// TwinCAT 3 PLC project V3_5
// Company: AQUAERO
// libraries:
//   Recipe Management,newest,System
//   VisuSymbols,3.5.10.0,System
//   Tc2_BA, * (Beckhoff Automation GmbH)
//   Tc2_Math, * (Beckhoff Automation GmbH)
//   Tc2_ModbusSrv, * (Beckhoff Automation GmbH)
//   Tc2_Standard, * (Beckhoff Automation GmbH)
//   Tc2_Standard, * (Beckhoff Automation GmbH)
//   Tc2_System, * (Beckhoff Automation GmbH)
//   Tc2_System, * (Beckhoff Automation GmbH)
//   Tc2_TcpIp, * (Beckhoff Automation GmbH)
//   Tc2_Utilities, * (Beckhoff Automation GmbH)
//   Tc3_BA_Common, * (Beckhoff Automation GmbH)
//   Tc3_Module, * (Beckhoff Automation GmbH)
//   Tc3_Module, * (Beckhoff Automation GmbH)
//   VisuDialogs, * (System)
// project tree:
//   Data types/ E_ClientServerSteps.TcDUT, ST_FrameFifoEntry.TcDUT
//   Global Variables/ GVL.TcGVL, GVL_1.TcGVL, TwinCAT_Configuration.TcGVL, Variablen_Konfiguration.TcGVL
//   / GlobalImagePool.TcGIPO (not stored), GlobalTextList.TcGTLO, Recipe Manager.TcRMO (not stored), Standard.TcTTO, Visualization Manager.TcVMO (not stored), VISU_TASK.TcTTO
//   POUs/ Average.TcPOU, Controller.TcPOU, FB_Blink.TcPOU, FB_PeerToPeer.TcPOU, SCL_MAIN.TcPOU, Meine_HYST.TcPOU
//   POUs/Helper POUs/ FB_FrameFifo.TcPOU, FB_LogFifo.TcPOU
//   Visualizations/ ImagePool.TcIPO (not stored), PID.TcVIS (not stored), Main.TcVIS (not stored), PID_alt.TcVIS (not stored), Layout.TcVIS (not stored), Heatreg.TcVIS (not stored), Sensors.TcVIS (not stored), Service.TcVIS (not stored), Testseite1.TcVIS (not stored), FRAME.TcVIS (not stored)
// real-time tasks:
//   TASK Standard: cycle T#10ms, priority 20, ADS port 350
//   TASK VISU_TASK: cycle T#200000us, priority 30, ADS port 351
//   TASK VISU_TASK1: cycle T#1ms, priority 1, ADS port 352

CONFIGURATION V3_5
    RESOURCE PLC ON TwinCAT3
        TASK Standard(INTERVAL := T#10ms, PRIORITY := 20);
        TASK VISU_TASK(INTERVAL := T#200000us, PRIORITY := 30);
        PROGRAM SCL_MAIN WITH Standard : SCL_MAIN;
        PROGRAM VisuElems_Visu_Prg WITH VISU_TASK : VisuElems.Visu_Prg;
    END_RESOURCE
END_CONFIGURATION

// ---- Data types/E_ClientServerSteps.TcDUT
TYPE E_ClientServerSteps :
(
	eUDP_STATE_IDLE		:= 0,
	eUDP_STATE_CREATE_START,
	eUDP_STATE_CREATE_WAIT,
	eUDP_STATE_SEND_START,
	eUDP_STATE_SEND_WAIT,
	eUDP_STATE_RECEIVE_START,
	eUDP_STATE_RECEIVE_WAIT,
	eUDP_STATE_CLOSE_START,
	eUDP_STATE_CLOSE_WAIT,
	eUDP_STATE_ERROR
);
END_TYPE

// ---- Data types/ST_FrameFifoEntry.TcDUT
TYPE ST_FrameFifoEntry :
STRUCT
	stRemoteAddr 	: ST_SockAddr;(* Remote address. String containing an (Ipv4) Internet Protocol dotted address and port number. *)
	sMessage		: T_MaxString;	(* UDP packet data *)
	r_Write_Example : REAL:=999;
	
	
	
END_STRUCT
END_TYPE

// ---- Global Variables/GVL.TcGVL






{attribute 'Tc2GvlVarNames'}
VAR_GLOBAL


(*_____________________________________________________________________________________________________________________________*)


	(*Ab hier Sind Globale Variablen Aquaero*)



	Main_Relais  AT%Q*:BOOL;
	Reset_M_R: BOOL;
	Set_M_R: BOOL;
	Reset_D_M: BOOL;
	Set_D_M: BOOL;
	Switch_OFF_Mainswitch: BOOL;









	(*Not-Aus Relais*)
	Feedback_Mainswitch AT%I*:BOOL;	(*EIngang NotAus-Relais*)
	Start_Mainswitch: BOOL;
	OUT_Mainswitch AT%Q*:BOOL;	(*Pulsausgang NotAus-Relais*)
	Mainswitch_OK: BOOL;
	ERROR_Mainswitch: BOOL;
	RESET_ERROR_Mainswitch: BOOL;
	Cabinet_OK: BOOL;
	VDC_24_OK AT%I*:BOOL;	(*Netzgerät OK*)

	VDC_OK: BOOL;











(* MODBUS *)

	mb_Input_Coils        : ARRAY [0..255] OF BOOL;
	mb_Output_Coils       : ARRAY [0..255] OF BOOL;
	mb_Input_Registers    : ARRAY [0..255] OF WORD;
	mb_Output_Registers   : ARRAY [0..255] OF WORD;



	Register_IN1: INT;
	Register_IN2: INT;
	Register_IN3: INT;
	Register_IN4: INT;
	Register_IN5: INT;
	Register_IN6: INT;
	Register_IN7: INT;
	Register_IN8: INT;
	Register_IN9: INT;
	Register_IN10: INT;



(*Regler_Kompressor Scroll*)


	Activate_controller_comp: BOOL;
	fRegelgroesse_comp: REAL;
	fSollwert_comp: REAL;				(*Ist zurzeit auf Sollert Dampfkammerdruck bezogen, der Kompressor ist das Stellglied*)
	fManual_controller_comp: REAL;
	Set_Manual_controller_comp: BOOL;
	fStellwert_comp: REAL;
	Reset_Controller_comp:BOOL;
	fKP_Controller_comp: REAL;
	fKI_Controller_comp: REAL;




(*Regler_Kompressor Klauenkolbenkomp.*)

	Activate_controller_Primaer_comp: BOOL;
	fRegelgroesse_Primaer_comp: REAL;
	fSollwert_Primaer_comp: REAL;
	fManual_controller_Primaer_comp: REAL;
	Set_Manual_controller_Primaer_comp: BOOL;
	fStellwert_Primaer_comp: REAL;
	Reset_Controller_Primaer_comp:BOOL;
	fKP_Controller_Primaer_comp: REAL:=1;
	fKI_Controller_Primaer_comp: REAL:=0.1;



(*Regler_Umdampfventi*)


	Activate_controller_V_Umdampf: BOOL;
	fRegelgroesse_V_Umdampf: REAL;
	fSollwert_V_Umdampf: REAL;				(*Ist zurzeit auf Sollert Dampfkammerdruck bezogen, der Kompressor ist das Stellglied*)
	fManual_controller_V_Umdampf: REAL;
	Set_Manual_controller_V_Umdampf: BOOL;
	fStellwert_V_Umdampf: REAL;
	Reset_Controller_V_Umdampf:BOOL;
	fKP_Controller_V_Umdampf: REAL;
	fKI_Controller_V_Umdampf: REAL;



(*Regler_Ventilator*)

	Activate_controller_Venti:  BOOL;
	fRegelgroesse_Venti: REAL;
	fSollwert_Venti: REAL;				(*Ist zurzeit auf Sollert Dampfkammerdruck bezogen, der Kompressor ist das Stellglied*)
	fManual_controller_Venti: REAL;
	Set_Manual_controller_Venti: BOOL;
	fStellwert_Venti: REAL;
	Reset_Controller_Venti:BOOL;
	fKP_Controller_Venti: REAL;
	fKI_Controller_Venti: REAL;




(*Regler_Nadelventil Swagelock*)



	Activate_controller_Needlevalve: BOOL;
	fRegelgroesse_NV: REAL;
	fSollwert_NV: REAL;				(*Ist zurzeit auf Sollert Dampfkammerdruck bezogen, der Kompressor ist das Stellglied*)
	fManual_controller_NV: REAL;
	Set_Manual_controller_NV: BOOL;
	fStellwert_NV: REAL;
	Reset_Controller_NV:BOOL;
	fKP_Controller_NV: REAL;
	fKI_Controller_NV: REAL;

	Sollwert_OUT_NV :INT;
	Istwert_IN_NV :INT;





	C_ADS: INT;
	C_DES: INT;




(*Ab hier: Sensorik und Aktorik des neuen Monstartors, oberhalb sind teils nicht verwendete Variablen!!*)





	T_Vor_WT_IN AT%I* : INT;
	T_Vor_WT:REAL;
	T_Vor_WT_Visu:REAL;
	T_nach_WT_IN AT%I* : INT;
	T_nach_WT:REAL;
	T_nach_WT_Visu:REAL;

	T_HE_Einduesung_Oben_IN AT%I* : INT;
	T_HE_Einduesung_Oben:REAL;
	T_HE_Einduesung_Oben_Visu:REAL;

	T_HE_Einduesung_Unten_IN AT%I* : INT;
	T_HE_Einduesung_Unten:REAL;
	T_HE_Einduesung_Unten_Visu:REAL;

	T_Einduesung_Unten_IN AT%I* : INT;
	T_Einduesung_Unten:REAL;
	T_Einduesung_Unten_Visu:REAL;

	T_Einduesung_Oben_IN AT%I* : INT;
	T_Einduesung_Oben:REAL;
	T_Einduesung_Oben_Visu:REAL;


	T_Absaugung_Oben_IN AT%I* : INT;
	T_Absaugung_Oben:REAL;
	T_Absaugung_Oben_Visu:REAL;

	T_Absaugung_Unten_IN AT%I* : INT;
	T_Absaugung_Unten:REAL;
	T_Absaugung_Unten_Visu:REAL;


	T_Vor_UmdampfLuefter_IN AT%I* : INT;
	T_Vor_UmdampfLuefter:REAL;
	T_Vor_UmdampfLuefter_Visu:REAL;

	T_Komp_Auslass_IN AT%I* : INT;
	T_Komp_Auslass:REAL;
	T_Komp_Auslass_Visu:REAL;

	T_Komp_Einlass_IN AT%I* : INT;
	T_Komp_Einlass:REAL;
	T_Komp_Einlass_Visu:REAL;


	T_Kond_Auslass_IN AT%I* : INT;
	T_Kond_Auslass:REAL;
	T_Kond_Auslass_Visu:REAL;

	T_DK_Oben_IN AT%I* : INT;
	T_DK_Oben:REAL;
	T_DK_Oben_Visu:REAL;

	T_DK_Mitte_IN AT%I* : INT;
	T_DK_Mitte:REAL;
	T_DK_Mitte_Visu:REAL;

	T_DK_Unten_IN AT%I* : INT;
	T_DK_Unten:REAL;
	T_DK_Unten_Visu:REAL;
	
	
	
	
	

	T_Mat_Auslass1_IN AT%I* : INT;
	T_Mat_Auslass1:REAL;
	T_Mat_Auslass1_Visu:REAL;
	T_Mat_Auslass2_IN AT%I* : INT;
	T_Mat_Auslass2:REAL;
	T_Mat_Auslass2_Visu:REAL;
	T_Mat_Auslass3_IN AT%I* : INT;
	T_Mat_Auslass3:REAL;
	T_Mat_Auslass3_Visu:REAL;
	T_Mat_Auslass4_IN AT%I* : INT;
	T_Mat_Auslass4:REAL;
	T_Mat_Auslass4_Visu:REAL;
	

	T_Mat_Auslass5_IN AT%I* : INT;
	T_Mat_Auslass5:REAL;
	T_Mat_Auslass5_Visu:REAL;
	T_Mat_Auslass6_IN AT%I* : INT;
	T_Mat_Auslass6:REAL;
	T_Mat_Auslass6_Visu:REAL;
	T_Mat_Auslass7_IN AT%I* : INT;
	T_Mat_Auslass7:REAL;
	T_Mat_Auslass7_Visu:REAL;
	T_Mat_Auslass8_IN AT%I* : INT;
	T_Mat_Auslass8:REAL;
	T_Mat_Auslass8_Visu:REAL;
	
	
	
	
	
	
	
	
	
	
	
	

	T_Komp_Gehaeuse_IN AT%I* : INT;
	T_Komp_Gehaeuse:REAL;
	T_Komp_Gehaeuse_Visu:REAL;


	T_DK_Band_oben1_IN AT%I* : INT;
	T_DK_Band_oben1:REAL;
	T_DK_Band_oben1_Visu:REAL;
	T_DK_Band_oben2_IN  : INT;
	T_DK_Band_oben2:REAL;
	T_DK_Band_oben2_Visu:REAL;
	T_DK_Band_oben3_IN AT%I* : INT;
	T_DK_Band_oben3:REAL;
	T_DK_Band_oben3_Visu:REAL;


	T_DK_Band_unten1_IN AT%I* : INT;
	T_DK_Band_unten1:REAL;
	T_DK_Band_unten1_Visu:REAL;
	T_DK_Band_unten2_IN : INT;
	T_DK_Band_unten2:REAL;
	T_DK_Band_unten2_Visu:REAL;
	T_DK_Band_unten3_IN AT%I* : INT;
	T_DK_Band_unten3:REAL;
	T_DK_Band_unten3_Visu:REAL;
	

	T_DK_Steigband1_IN AT%I* : INT;
	T_DK_Steigband1:REAL;
	T_DK_Steigband1_Visu:REAL;
	T_DK_Steigband2_IN AT%I* : INT;
	T_DK_Steigband2:REAL;
	T_DK_Steigband2_Visu:REAL;
	T_DK_Steigband3_IN AT%I* : INT;
	T_DK_Steigband3:REAL;
	T_DK_Steigband3_Visu:REAL;
	T_DK_Steigband4_IN AT%I* : INT;
	T_DK_Steigband4:REAL;
	T_DK_Steigband4_Visu:REAL;

	
	
	
	
	
	


	Temp_Heatmatt1_IN  AT%I* : INT;
	Temp_Heatmatt2_IN  AT%I* : INT;
	Temp_Heatmatt3_IN  AT%I* : INT;
	Temp_Heatmatt4_IN  AT%I* : INT;
	Temp_Heatmatt5_IN  AT%I* : INT;
	Temp_Heatmatt6_IN  AT%I* : INT;
	Temp_Heatmatt7_IN  AT%I* : INT;
	Temp_Heatmatt8_IN  AT%I* : INT;
	Temp_Heatmatt9_IN  AT%I* : INT;
	Temp_Heatmatt10_IN  AT%I* : INT;


	

	Temp_Heatmatt1 : INT;
	Temp_Heatmatt2 : INT;
	Temp_Heatmatt3 : INT;
	Temp_Heatmatt4 : INT;
	Temp_Heatmatt5 : INT;
	Temp_Heatmatt6 : INT;
	Temp_Heatmatt7 : INT;
	Temp_Heatmatt8 : INT;
	Temp_Heatmatt9 : INT;
	Temp_Heatmatt10 : INT;

	Temp_compressor_Self : INT;




	P_Vor_WT_IN AT%I* : INT;
	P_Vor_WT:REAL;
	P_Vor_WT_Visu:REAL;


	P_Durchfluss_IN  : INT;
	P_Durchfluss:REAL;
	P_Durchfluss_Visu:REAL;



	P_Komp_Einlass_IN AT%I* : INT;
	P_Komp_Einlass:REAL;
	P_Komp_Einlass_Visu:REAL;


	P_Komp_Auslass_IN AT%I* : INT;
	P_Komp_Auslass:REAL;
	P_Komp_Auslass_Visu:REAL;


	W_Kond_Wasser_IN AT%I* : INT;
	W_Kond_Wasser:REAL;
	W_Kond_Wasser_Visu:REAL;



	O2_IN AT%I* : INT;
	O2:REAL;
	O2_Visu:REAL;

	

	PTC_IN:BOOL;
	Motor_HOT:BOOL;

	Switch_Heat_group1:BOOL;
	Switch_Heat_group2:BOOL;
	Switch_Heat_group3:BOOL;
	Start_Auto_Export: BOOL;
	Start_Auto_Export_OUT: BOOL;




	(* Diverses (teils noch von älterenb Programmfunktionen*)

	Pulse2_set_manu:BOOL;
	Enable_Pulsgen2 :BOOL;
	T_Pulstime_Pulsegen2: INT:=3;
	T_HI_Pulsegen2: INT:=20;
	Valve_YB7:BOOL;












(*Strom und Energiemessung*)


	(*Current_IN_HZE_Auffangbecken_L1 AT%I*:INT;
	Current_IN_HZE_Auffangbecken_L2 AT%I*:INT;
	Current_IN_HZE_Auffangbecken_L3 AT%I*:INT;*)

	Current_IN_HEAT_Reg_1 AT%I*:INT;
	Current_IN_HEAT_Reg_2 AT%I*:INT;
	Current_IN_HEAT_Reg_3 AT%I*:INT;
	Current_IN_HEAT_Reg_4 AT%I*:INT;
	Current_IN_HEAT_Reg_5 AT%I*:INT;
	Current_IN_HEAT_Reg_6 AT%I*:INT;
	Current_IN_HEAT_Reg_7 AT%I*:INT;
	Current_IN_HEAT_Reg_8 AT%I*:INT;
	Current_IN_Compressor_L1 AT%I*:INT;
	Current_IN_Compressor_L2 AT%I*:INT;
	Current_IN_Compressor_L3 AT%I*:INT;
	Current_IN_SteamFan_L1 AT%I*:INT;
	Current_IN_SteamFan_L2 AT%I*:INT;
	Current_IN_SteamFan_L3 AT%I*:INT;
	Current_IN_Fan_L1 AT%I*:INT;
	Current_IN_Fan_L2 AT%I*:INT;
	Current_IN_Fan_L3 AT%I*:INT;
	Current_IN_Complete_L1 AT%I*:INT;
	Current_IN_Complete_L2 AT%I*:INT;
	Current_IN_Complete_L3 AT%I*:INT;



	

	Current_OUT_SteamVenti_L1:REAL;
	Current_OUT_SteamVenti_L2:REAL;
	Current_OUT_SteamVenti_L3:REAL;
	Current_OUT_HEAT_Reg_1:REAL;
	Current_OUT_HEAT_Reg_2:REAL;
	Current_OUT_HEAT_Reg_3:REAL;
	Current_OUT_HEAT_Reg_4:REAL;
	Current_OUT_HEAT_Reg_5:REAL;
	Current_OUT_HEAT_Reg_6:REAL;
	Current_OUT_HEAT_Reg_7:REAL;
	Current_OUT_HEAT_Reg_8:REAL;






	Current_OUT_Compressor_L1 :REAL;
	Current_OUT_Compressor_L2 :REAL;
	Current_OUT_Compressor_L3 :REAL;

	Current_OUT_AdsorbtionsVenti_L1 :REAL;
	Current_OUT_AdsorbtionsVenti_L2 :REAL;
	Current_OUT_AdsorbtionsVenti_L3 :REAL;
	Current_OUT_Fan_L1:REAL;
	Current_OUT_Fan_L2 :REAL;
	Current_OUT_Fan_L3:REAL;
	Current_OUT_Complete_L1 :REAL;
	Current_OUT_Complete_L2 :REAL;
	Current_OUT_Complete_L3 :REAL;






	(*Energy_IN_HZE_Auffangbecken_L1 AT%I*:INT;
	Energy_IN_HZE_Auffangbecken_L2 AT%I*:INT;
	Energy_IN_HZE_Auffangbecken_L3 AT%I*:INT;*)

	(*
	Energy_IN_HEAT_Reg_1 AT%I*:INT;
	Energy_IN_HEAT_Reg_2 AT%I*:INT;
	Energy_IN_HEAT_Reg_3 AT%I*:INT;
	Energy_IN_HEAT_Reg_4 AT%I*:INT;
	Energy_IN_Compressor_L1 AT%I*:INT;
	Energy_IN_Compressor_L2 AT%I*:INT;
	Energy_IN_Compressor_L3 AT%I*:INT;
	Energy_IN_SteamFan_L1 AT%I*:INT;
	Energy_IN_SteamFan_L2 AT%I*:INT;
	Energy_IN_SteamFan_L3 AT%I*:INT;
	Energy_IN_Fan_L1 AT%I*:INT;
	Energy_IN_Fan_L2 AT%I*:INT;
	Energy_IN_Fan_L3 AT%I*:INT;
	Energy_IN_Complete_L1 AT%I*:INT;
	Energy_IN_Complete_L2 AT%I*:INT;
	Energy_IN_Complete_L3 AT%I*:INT;*)

	
	
	

	Energy_OUT_HZE_Auffangbecken_L1:REAL;
	Energy_OUT_HZE_Auffangbecken_L2:REAL;
	Energy_OUT_HZE_Auffangbecken_L3:REAL;

	Energy_OUT_HEAT_Reg_1:REAL;
	Energy_OUT_HEAT_Reg_2:REAL;
	Energy_OUT_HEAT_Reg_3:REAL;
	Energy_OUT_HEAT_Reg_4:REAL;
	Energy_OUT_HEAT_Reg_5:REAL;
	Energy_OUT_HEAT_Reg_6:REAL;
	Energy_OUT_HEAT_Reg_7:REAL;
	Energy_OUT_HEAT_Reg_8:REAL;





	Energy_OUT_Compressor_L1 :REAL;
	Energy_OUT_Compressor_L2 :REAL;
	Energy_OUT_Compressor_L3 :REAL;
	Energy_OUT_SteamFan_L1 :REAL;
	Energy_OUT_SteamFan_L2 :REAL;
	Energy_OUT_SteamFan_L3 :REAL;
	Energy_OUT_Fan_L1:REAL;
	Energy_OUT_Fan_L2 :REAL;
	Energy_OUT_Fan_L3:REAL;
	Energy_OUT_Complete_L1 :REAL;
	Energy_OUT_Complete_L2 :REAL;
	Energy_OUT_Complete_L3 :REAL;






(*_________Frequence_Converter_Groups and controls*)

	Compressor_ON AT%Q* : BOOL;
	Compressor_Switch_ON AT%Q* : BOOL;
	Compressor_OK AT%I* : BOOL;
	Compressor_Circuit_breaker AT%I* : BOOL;
	Compressor_Setpoint_OUT AT%Q* : INT;
	Setpoint_Compressor_IN: INT;
	Setpoint_Compressor_Auto: INT;
	Setpoint_Compressor_Visu: INT;
	Compressor_Actual_Turn_IN AT%I* : INT;
	Compressor_Actual_Turn: REAL;
	Limit_Temp_Compressor: INT:=100;
	Temp_compressor_OK: BOOL;
	T_Ueberwachung_scroll_comp AT%I* : INT;


	Compressor_cooling  : BOOL;
	Compressor_cooling_manu  : BOOL;
	Compressor_cooling_auto : BOOL;
	Compressor_Switch_ON_Manu: BOOL;
	Compressor_ON_Manu: BOOL;
	Compressor_PT100_value AT%I* : INT;
	Compressor_PT100_error AT%I* : BOOL;






	(*
	PRIMAER_Comp_ON AT%Q* : BOOL;
	PRIMAER_Comp_OK AT%I* : BOOL;
	PRIMAER_Comp_Setpoint_OUT AT%Q* : INT;
	Setpoint_PRIMAER_Comp_IN: INT;
	Setpoint_PRIMAER_Comp_Auto: INT;
	Setpoint_PRIMAER_Comp_Visu: INT;
	PRIMAER_Comp_Actual_Turn_IN AT%I* : INT;
	PRIMAER_Comp_Actual_Turn: REAL;
	Temp_PRIMAER_Comp_OK: BOOL;
	PRIMAER_Comp_Switch_ON_Manu: BOOL;
	PRIMAER_Comp_ON_Manu: BOOL;
	*)



	Fan_ON  : BOOL;
	Fan_OK  : BOOL;
	Setpoint_Fan_Auto: INT;
	Setpoint_Fan_Visu: INT;
	Setpoint_Fan_OUT  : INT;
	Setpoint_Fan_IN: INT;
	Fan_Actual_Turn_IN  : INT;
	Fan_Actual_Turn  : REAL;
	FAN_Switch_ON  : BOOL;
	FAN_Switch_ON_Manu: BOOL;
	FAN_ON_Manu: BOOL;



	SteamFan_ON AT%Q* : BOOL;
	SteamFan_OK :BOOL ;(* Zurzeit nicht einlesbar AT%I* : BOOL;*)
	Setpoint_SteamFan_Auto: INT;
	Setpoint_SteamFan_Visu: INT;
	Setpoint_SteamFan_OUT AT%Q* : INT;
	Setpoint_SteamFan_IN: INT;
	SteamFan_Actual_Turn_IN AT%I* : INT;
	SteamFan_Actual_Turn  : REAL;
	SteamFAN_Switch_ON AT%Q* : BOOL;
	SteamFAN_Switch_ON_manu:BOOL;
	SteamFan_ON_manu:BOOL;
	Setpoint_SteamFan_manu:INT;
	SteamFan_PTC_IN AT%I* : BOOL;
	SteamFan_PTC_Error AT%I* : BOOL;



	M_Belts_ON AT%Q* : BOOL;
	M_Belts_OK AT%I* : BOOL;
	Setpoint_M_Belts_Auto: INT;
	Setpoint_M_Belts_Visu: INT;
	Setpoint_M_Belts_OUT AT%Q* : INT;
	Setpoint_M_Belts_IN: INT;
	M_Belts_Actual_Turn_IN AT%I* : INT;
	M_Belts_Actual_Turn  : REAL;
	M_Belts_Switch_ON AT%Q* : BOOL;
	M_Belts_Switch_ON_Manu: BOOL;
	M_Belts_ON_Manu: BOOL;
	Activate_controller_M_Belts:BOOL;
	fStellwert_M_Belts:REAL;


	M_Belt_Feeder_ON AT%Q* : BOOL;
	M_Belt_Feeder_OK AT%I* : BOOL;
	Setpoint_M_Belt_Feeder_Auto: INT;
	Setpoint_M_Belt_Feeder_Visu: INT;
	Setpoint_M_Belt_Feeder_OUT AT%Q* : INT;
	Setpoint_M_Belt_Feeder_IN: INT;
	M_Belt_Feeder_Actual_Turn_IN AT%I* : INT;
	M_Belt_Feeder_Actual_Turn  : REAL;
	M_Belt_Feeder_Switch_ON AT%Q* : BOOL;
	M_Belt_Feeder_Switch_ON_Manu: BOOL;
	M_Belt_Feeder_ON_Manu: BOOL;
	Activate_controller_M_Belt_Feeder:BOOL;
	fStellwert_M_Belt_Feeder:REAL;


	Steamgenerator : BOOL;
	Steamgenerator_manu: BOOL;
	Steamgenerator_auto: BOOL;



(*_________Frequence_Converter_Groups AND controls*)
















	(*OUT_______BOOL____________*)



	

	V_Dampf_nach_Komp  AT%Q* : BOOL ;
	V_Dampf_nach_Komp_negiert  AT%Q* : BOOL;
	V_Nach_WT  AT%Q* : BOOL;
	V_Entlueftung_1 AT%Q* : BOOL;
	V_Entlueftung_2 AT%Q* : BOOL;
	V_Global_Res_3 AT%Q* : BOOL;
	V_Global_Res_4 AT%Q* : BOOL;
	V_Global_Res_5 AT%Q* : BOOL;




	Heizelement_Auffangbecken_Mainswitch: BOOL;



	Heat_matt_Group1_1_4 :BOOL;
	Heat_matt_Group2_5_8 :BOOL;
	Heat_matt_Group3_9_10: BOOL;

	Heat_matt1 : BOOL;
	Heat_matt2 : BOOL;
	Heat_matt3 : BOOL;
	Heat_matt4 : BOOL;
	Heat_matt5 : BOOL;
	Heat_matt6 : BOOL;
	Heat_matt7 : BOOL;
	Heat_matt8 : BOOL;
	Heat_matt9 : BOOL;
	Heat_matt10 : BOOL;


	Heat_Matt1_OK_for_heat:BOOL;
	Heat_Matt2_OK_for_heat:BOOL;
	Heat_Matt3_OK_for_heat:BOOL;
	Heat_Matt4_OK_for_heat:BOOL;
	Heat_Matt5_OK_for_heat:BOOL;
	Heat_Matt6_OK_for_heat:BOOL;
	Heat_Matt7_OK_for_heat:BOOL;
	Heat_Matt8_OK_for_heat:BOOL;
	Heat_Matt9_OK_for_heat:BOOL;
	Heat_Matt10_OK_for_heat:BOOL;
	Heat_Matt11_OK_for_heat: BOOL;




	HEAT_Reg_Mainswitch_OUT : BOOL;


	HEAT_Reg_1_OUT AT%Q* : BOOL;
	HEAT_Reg_2_OUT AT%Q* : BOOL;
	HEAT_Reg_3_OUT AT%Q* : BOOL;
	HEAT_Reg_4_OUT AT%Q* : BOOL;
	HEAT_Reg_5_OUT AT%Q* : BOOL;
	HEAT_Reg_6_OUT AT%Q* : BOOL;
	HEAT_Reg_7_OUT AT%Q* : BOOL;
	HEAT_Reg_8_OUT AT%Q* : BOOL;






	V_Nach_WT_negiert: BOOL;
	V_Wasserauslass_negiert: BOOL;
	V_Entlueftung_1_negiert: BOOL;
	V_Global_Res_5_negiert: BOOL;
	V_Global_Res_4_negiert: BOOL;
	V_Global_Res_3_negiert: BOOL;
	V_Entlueftung_2_negiert: BOOL;







	(*AUTO_____________BOOL_____________*)




	(*neuere Aktoren von MS2*)

	V_Dampf_nach_Komp_auto : BOOL:=FALSE;
	V_Nach_WT_auto:BOOL:=FALSE;
	V_Entlueftung_1_auto : BOOL;
	V_Entlueftung_2_auto : BOOL:=FALSE;
	V_Global_Res_3_auto : BOOL:=FALSE;
	V_Global_Res_4_auto : BOOL:=FALSE;
	V_Global_Res_5_auto : BOOL;



	Heat_matt1_auto: BOOL;
	Heat_matt2_auto: BOOL;
	Heat_matt3_auto: BOOL;
	Heat_matt4_auto: BOOL;
	Heat_matt5_auto: BOOL;
	Heat_matt6_auto: BOOL;
	Heat_matt8_auto: BOOL;
	Heat_matt7_auto:BOOL;
	Heat_matt9_auto: BOOL;
	Heat_matt10_auto: BOOL;

	Heat_matt_Group1_1_4_auto: BOOL;
	Heat_matt_Group2_5_8_auto: BOOL;
	Heat_matt_Group3_9_10_auto: BOOL;


	HEAT_Reg_Mainswitch_Auto:BOOL;

	HEAT_Reg_1_Auto: BOOL;
	HEAT_Reg_2_Auto: BOOL;
	HEAT_Reg_3_Auto: BOOL;
	HEAT_Reg_4_Auto: BOOL;
	HEAT_Reg_5_Auto: BOOL;
	HEAT_Reg_6_Auto: BOOL;
	HEAT_Reg_7_Auto: BOOL;
	HEAT_Reg_8_Auto: BOOL;







	(*MANU____________BOOL___________*)


	(*neuere Aktoren von MS2*)


	V_Dampf_nach_Komp_manu : BOOL:=FALSE;
	V_Nach_WT_manu : BOOL:=FALSE;
	V_Entlueftung_1_manu : BOOL:=FALSE;
	V_Entlueftung_2_manu : BOOL;
	V_Global_Res_3_manu : BOOL;
	V_Global_Res_4_manu: BOOL:=FALSE;
	V_Global_Res_5_manu : BOOL;




	Heat_matt1_manu: BOOL;
	Heat_matt2_manu: BOOL;
	Heat_matt3_manu: BOOL;
	Heat_matt4_manu: BOOL;
	Heat_matt5_manu: BOOL;
	Heat_matt6_manu: BOOL;
	Heat_matt7_manu: BOOL;
	Heat_matt8_manu: BOOL;
	Heat_matt9_manu: BOOL;
	Heat_matt10_manu: BOOL;



	HEAT_Reg_Mainswitch_Manu:BOOL;


	HEAT_Reg_1_Manu: BOOL;
	HEAT_Reg_2_Manu: BOOL;
	HEAT_Reg_3_Manu: BOOL;
	HEAT_Reg_4_Manu: BOOL;
	HEAT_Reg_5_Manu: BOOL;
	HEAT_Reg_6_Manu: BOOL;
	HEAT_Reg_7_Manu: BOOL;
	HEAT_Reg_8_Manu: BOOL;





(*________________________________________________________________ENDE_MANU_Vars________________________________*)


















	V_Entlueftung_1_Reset:BOOL;
	V_Entlueftung_2_Reset:BOOL;
	V_Global_Res_3_Reset:BOOL;
	V_Global_Res_4_Reset:BOOL;
	V_Global_Res_5_Reset:BOOL;
	V_Dampf_nach_Komp_Reset:BOOL;
	V_Nach_WT_Reset:BOOL;


	V_Entlueftung_1_String:STRING;
	V_Entlueftung_2_String:STRING;
	V_Global_Res_3_String:STRING;
	V_Global_Res_4_String:STRING;
	V_Global_Res_5_String:STRING;
	V_Dampf_nach_Komp_String:STRING;
	V_NACH_WT_String:STRING;


	V_Entlueftung_1_Reset_Sequence:BOOL;
	V_Entlueftung_2_Reset_Sequence:BOOL;
	V_Global_Res_3_Reset_Sequence:BOOL;
	V_Global_Res_4_Reset_Sequence:BOOL;
	V_Global_Res_5_Reset_Sequence:BOOL;
	V_Dampf_nach_Komp_Reset_Sequence:BOOL;
	V_NACH_WT_Reset_Sequence:BOOL;


	V_Entlueftung_1_Sequence:BOOL;
	V_Entlueftung_2_Sequence:BOOL;
	V_Global_Res_3_Sequence:BOOL;
	V_Global_Res_4_Sequence:BOOL;
	V_Global_Res_5_Sequence:BOOL;
	V_Dampf_nach_Komp_Sequence:BOOL;
	V_NACH_WT_Sequence:BOOL;



	VE_K2_71:BOOL;
	VE_K2_73:BOOL;











	LED_RED_OUT AT%Q* :BOOL;
	LED_RED_VISU: BOOL;
	LED_RED_auto: BOOL;

	LED_green_OUT AT%Q* :BOOL;
	LED_green_VISU: BOOL;
	LED_green_auto: BOOL;

	LED_yellow_OUT AT%Q* :BOOL;
	LED_yellow_VISU: BOOL;
	LED_yellow_auto: BOOL;

	LED_white_OUT AT%Q* :BOOL;
	LED_white_VISU: BOOL;
	LED_white_auto: BOOL;


	All_Heater_on_auto:BOOL;













	Control_Manu: BOOL;
	Control_Manu_active: BOOL;
	Reset_man: BOOL;
	Control_Auto: BOOL;
	Control_Auto_active: BOOL;
	Reset_auto: BOOL;


	Control_ADS: BOOL;
	ADS_active: BOOL;
	Reset_ADS: BOOL;
	Control_DES: BOOL;
	DES_active: BOOL;
	Reset_DES: BOOL;




	P_Cabinet_Underlimit: INT:=700;	(*mbar*)







	(*Reglerbausteine für PWM Ausgänge*)


	(*Parameter*)

	//Als Testzweck draussen
	(*stParams: ST_CTRL_2POINT_PWM_ADAPTIVE_PARAMS;
	Heat_REG1_CTRL_PWM:FB_CTRL_2POINT_PWM_ADAPTIVE;
	Heat_REG2_CTRL_PWM:FB_CTRL_2POINT_PWM_ADAPTIVE;
	Heat_REG3_CTRL_PWM:FB_CTRL_2POINT_PWM_ADAPTIVE;
	Heat_REG4_CTRL_PWM:FB_CTRL_2POINT_PWM_ADAPTIVE;
	Heat_REG5_CTRL_PWM:FB_CTRL_2POINT_PWM_ADAPTIVE;
	Heat_REG6_CTRL_PWM:FB_CTRL_2POINT_PWM_ADAPTIVE;
	Heat_REG7_CTRL_PWM:FB_CTRL_2POINT_PWM_ADAPTIVE;
	Heat_REG8_CTRL_PWM:FB_CTRL_2POINT_PWM_ADAPTIVE;*)



	
	
	
	(*Heat_EinschraubHZK1_CTRL_PWM:FB_CTRL_2POINT_PWM_ADAPTIVE;
	Heat_EinschraubHZK2_CTRL_PWM:FB_CTRL_2POINT_PWM_ADAPTIVE;
	Heat_EinschraubHZK3_CTRL_PWM:FB_CTRL_2POINT_PWM_ADAPTIVE;
	Heat_REG_Comp:FB_CTRL_2POINT_PWM_ADAPTIVE;*)



	(*INPUTS*)

	fSetpointValue1			:FLOAT:=20;	(*Heizregister 1-4 zurzeit alls Gruppe (oben) *)
	fSetpointValue2			:FLOAT:=20;	(*Heizregister 5-8 zurzeit alls Gruppe (oben) *)

	fSetpointValue3			:FLOAT:=20;
	fSetpointValue4			:FLOAT:=20;

	fSetpointValue5			:FLOAT:=20;	(* Setpoints 5-7 waren ehemals EInschraubheizkörper*)
	fSetpointValue6			:FLOAT:=20;
	fSetpointValue7			:FLOAT:=20;

	fSetpointValue8			:FLOAT:=20;


	
	//Als Testzweck draussen
	(*
	fManSyncValue			:FLOAT;					(* input value for the manual mode or the sync request *)
	bSync					: BOOL;							(* rising edge set the output to the fManSyncValue *)
	eMode					: E_CTRL_MODE;					(* sets the mode of the function block *)
	bHold					: BOOL;							(* hold the internal integrator *)

	eState				: E_CTRL_STATE;
	eErrorId				: E_CTRL_ERRORCODES;		(* error code *)
	bError				: BOOL;*)
	
	
	


	(*OUTPUTS*)

	fPWMDutyCycle1		:FLOAT;					(* fOut reached the max or min limit *)
	fPWMDutyCycle2		:FLOAT;				(* fOut reached the max or min limit *)
	fPWMDutyCycle3		:FLOAT;						(* fOut reached the max or min limit *)
	fPWMDutyCycle4		:FLOAT;
	fPWMDutyCycle5		:FLOAT;
	fPWMDutyCycle6		:FLOAT;
	fPWMDutyCycle7		:FLOAT;
	fPWMDutyCycle8		:FLOAT;











	bManuHeat_REG1_CTRL: BOOL;
	bAuto_Heat_REG1_CTRL: BOOL;
	bManuHeat_REG2_CTRL: BOOL;
	bAuto_Heat_REG2_CTRL: BOOL;
	bManuHeat_REG3_CTRL: BOOL;
	bAuto_Heat_REG3_CTRL: BOOL;
	bManuHeat_REG4_CTRL: BOOL;
	bAuto_Heat_REG4_CTRL: BOOL;

	bManuHeat_REG5_CTRL: BOOL;
	bAuto_Heat_REG5_CTRL: BOOL;
	bManuHeat_REG6_CTRL: BOOL;
	bAuto_Heat_REG6_CTRL: BOOL;
	bManuHeat_REG7_CTRL: BOOL;
	bAuto_Heat_REG7_CTRL: BOOL;
	bManuHeat_REG8_CTRL: BOOL;
	bAuto_Heat_REG8_CTRL: BOOL;

	T_Limit_Heatreg_top: REAL:=200.0;
	T_Limit_Heatreg_bottom: REAL:=200.0;









	(*bManu_Heat_EinschraubHZK1_CTRL: BOOL;
	bAuto_Heat_EinschraubHZK1_CTRL: BOOL;
	bManu_Heat_EinschraubHZK2_CTRL: BOOL;
	bAuto_Heat_EinschraubHZK2_CTRL: BOOL;
	bManu_Heat_EinschraubHZK3_CTRL: BOOL;
	bAuto_Heat_EinschraubHZK3_CTRL: BOOL;
	bManu_Heat_REG_Comp: BOOL;
	bAuto_Heat_REG_Comp: BOOL;*)


	 Ctr_Manu: BOOL;
	 Ctr_Auto: BOOL;
	 Ctr_Reset: BOOL;


	 Ctr_Manu_active: BOOL;
	 Ctr_Auto_active: BOOL;
	 Ctr_Reset_active: BOOL;



	OKRange_Ctrl:FLOAT:=2; (*%*)

	Step_Size_Ctr_PWM:FLOAT:=5;	(*%*)

	Force_Range_ON: FLOAT:=5;	(*Celcius*)


(*Bis Hier ControlParameter*)


































	(*Modbus Server Variables*)

	ipAddr 			:	STRING(15) :='192.168.100.66';	(*Pokeys*)
	(*M0 AT%MB0		:	ARRAY [0..3] OF WORD;*)
	nValue			: 	ARRAY [0..6] OF WORD ;
	bWriteRegs		:  	BOOL;
	PWM_duty_cycle: UINT;
	nTCPPort 		: UINT:= 503;
	nUnitID 		: BYTE:=16#FF;
	bBUSY 		: BOOL;
	bbError 		: BOOL;
	nErrId 		: UDINT;





	XY: INT;
	 C_val1:WORD;
	Valve_YB9: BOOL;
	Valve_YB10: BOOL;
	Valvematrix2: BYTE;


	Reset_Sequence: BOOL;


	Hyst_low_LIM_Heatmatt: INT:=120;
	Hyst_high_LIM_Heatmatt: INT:=140;
	Case_Schritt: INT;

	Start_Puls_Valves: BOOL;
	Start_Puls_Valves_out: BOOL;



	(*____GUEST VAR___________*)







	(*____GUEST VAR___________*)




	Poti_Istwert_NV: REAL;
	High_Limit_Poti_Istwert_NV: REAL;
	Low_Limit_Poti_Istwert_NV: REAL;


	P_Saetigung: REAL;
	T_Saetigung: REAL;

	Ps_311: REAL;
	Ps_26: REAL;
	Ps_28: REAL;
	Ps_23: REAL;

	RelP_TM: REAL;
	RelP_TM2: REAL;
	RelP_WT: REAL;
	RelP_Out: REAL;

	testvar: REAL;
	Konstant1: REAL:=2;
	nErrorStatus_comp: UINT;
	nErrorStatus_NV: UINT;
	
	
	fKP_Controller_Heatmatt1: LREAL;
	fKI_Controller_Heatmatt1: LREAL;
	nErrorStatus_Heatmatt1: UINT;
	
	
	fKP_Controller_Heatmatt2: LREAL;
	fKI_Controller_Heatmatt2: LREAL;
	nErrorStatus_Heatmatt2: UINT;
	
	
	fKP_Controller_Heatmatt3: LREAL;
	fKI_Controller_Heatmatt3: LREAL;
	nErrorStatus_Heatmatt3: UINT;
	
	
	fKP_Controller_Heatmatt4: LREAL;
	fKI_Controller_Heatmatt4: LREAL;
	nErrorStatus_Heatmatt4: UINT;
	
	
	
	
	
	
	

	
	
	
	T_Monitor_Heatreg1: REAL;
	T_Limit_Heatreg: REAL;
	T_Monitor_Heatreg2: REAL;
	
	
	
	
	//Für Webbrowser:
	
	SurlAdress:STRING:='www.psi.ch';
	bBack:BOOL;
	bForward:BOOL;
	bShow:BOOL;
	
	aArray_Histogram:ARRAY[0..100]OF INT;
	
	
	counup_Array: INT;
	counup_Array_OUT: INT;
	Istwert_IN_NV_OUT: REAL;
	fTemp_mean_belt_top: REAL;
	fTemp_mean_belt_bottom: REAL;
	Reset_heatreg_top: BOOL;
	Reset_heatreg_bottom: BOOL;
	Reset_heatreg_compressor: BOOL;
	OK_For_HEAT_WHILE_FAN_IS_ON: BOOL;
END_VAR




//Für UDP Kommunikation


VAR_GLOBAL CONSTANT
	PLCPRJ_BUFFER_SIZE					: UDINT := 1000;(* Max. internal fifo/receiver buffer size *)

	(* Some project specific error codes *)
	PLCPRJ_ERROR_SENDFIFO_OVERFLOW		: UDINT := 16#8103;
	PLCPRJ_ERROR_RECFIFO_OVERFLOW		: UDINT := 16#8104;
END_VAR

// ---- Global Variables/GVL_1.TcGVL
VAR_GLOBAL
	
(*Ab hier: Sensorik und Aktorik des neuen Monstartors, oberhalb sind teils nicht verwendete Variablen!!*)


Scope_T_Vor_WT_IN AT%I* : INT;
Scope_T_Vor_WT:REAL;
Scope_T_Vor_WT_Visu:REAL;
Scope_T_nach_WT_IN AT%I* : INT;
Scope_T_nach_WT:REAL;
Scope_T_nach_WT_Visu:REAL;
Scope_T_HE_Einduesung_Oben_IN AT%I* : INT;
Scope_T_HE_Einduesung_Oben:REAL;
Scope_T_HE_Einduesung_Oben_Visu:REAL;
Scope_T_HE_Einduesung_Unten_IN AT%I* : INT;
Scope_T_HE_Einduesung_Unten:REAL;
Scope_T_HE_Einduesung_Unten_Visu:REAL;
Scope_T_Einduesung_Unten_IN AT%I* : INT;
Scope_T_Einduesung_Unten:REAL;
Scope_T_Einduesung_Unten_Visu:REAL;
Scope_T_Einduesung_Oben_IN AT%I* : INT;
Scope_T_Einduesung_Oben:REAL;
Scope_T_Einduesung_Oben_Visu:REAL;
Scope_T_Absaugung_Oben_IN AT%I* : INT;
Scope_T_Absaugung_Oben:REAL;
Scope_T_Absaugung_Oben_Visu:REAL;
Scope_T_Absaugung_Unten_IN AT%I* : INT;
Scope_T_Absaugung_Unten:REAL;
Scope_T_Absaugung_Unten_Visu:REAL;
Scope_T_Vor_UmdampfLuefter_IN AT%I* : INT;
Scope_T_Vor_UmdampfLuefter:REAL;
Scope_T_Vor_UmdampfLuefter_Visu:REAL;
Scope_T_Komp_Auslass_IN AT%I* : INT;
Scope_T_Komp_Auslass:REAL;
Scope_T_Komp_Auslass_Visu:REAL;
Scope_T_Komp_Einlass_IN AT%I* : INT;
Scope_T_Komp_Einlass:REAL;
Scope_T_Komp_Einlass_Visu:REAL;
Scope_T_Kond_Auslass_IN AT%I* : INT;
Scope_T_Kond_Auslass:REAL;
Scope_T_Kond_Auslass_Visu:REAL;
Scope_T_DK_Oben_IN AT%I* : INT;
Scope_T_DK_Oben:REAL;
Scope_T_DK_Oben_Visu:REAL;
Scope_T_DK_Mitte_IN AT%I* : INT;
Scope_T_DK_Mitte:REAL;
Scope_T_DK_Mitte_Visu:REAL;
Scope_T_DK_Unten_IN AT%I* : INT;
Scope_T_DK_Unten:REAL;
Scope_T_DK_Unten_Visu:REAL;
Scope_T_Mat_Auslass1_IN AT%I* : INT;
Scope_T_Mat_Auslass1:REAL;
Scope_T_Mat_Auslass1_Visu:REAL;
Scope_T_Mat_Auslass2_IN AT%I* : INT;
Scope_T_Mat_Auslass2:REAL;
Scope_T_Mat_Auslass2_Visu:REAL;
Scope_T_Mat_Auslass3_IN AT%I* : INT;
Scope_T_Mat_Auslass3:REAL;
Scope_T_Mat_Auslass3_Visu:REAL;
Scope_T_Mat_Auslass4_IN AT%I* : INT;
Scope_T_Mat_Auslass4:REAL;
Scope_T_Mat_Auslass4_Visu:REAL;
Scope_T_Komp_Gehaeuse_IN AT%I* : INT;
Scope_T_Komp_Gehaeuse:REAL;
Scope_T_Komp_Gehaeuse_Visu:REAL;
Scope_T_DK_Band_oben1_IN AT%I* : INT;
Scope_T_DK_Band_oben1:REAL;
Scope_T_DK_Band_oben1_Visu:REAL;
Scope_T_DK_Band_oben2_IN AT%I* : INT;
Scope_T_DK_Band_oben2:REAL;
Scope_T_DK_Band_oben2_Visu:REAL;
Scope_T_DK_Band_oben3_IN AT%I* : INT;
Scope_T_DK_Band_oben3:REAL;
Scope_T_DK_Band_oben3_Visu:REAL;
Scope_T_DK_Band_unten1_IN AT%I* : INT;
Scope_T_DK_Band_unten1:REAL;
Scope_T_DK_Band_unten1_Visu:REAL;
Scope_T_DK_Band_unten2_IN AT%I* : INT;
Scope_T_DK_Band_unten2:REAL;
Scope_T_DK_Band_unten2_Visu:REAL;
Scope_T_DK_Band_unten3_IN AT%I* : INT;
Scope_T_DK_Band_unten3:REAL;
Scope_T_DK_Band_unten3_Visu:REAL;
Scope_T_DK_Steigband1_IN AT%I* : INT;
Scope_T_DK_Steigband1:REAL;
Scope_T_DK_Steigband1_Visu:REAL;
Scope_T_DK_Steigband2_IN AT%I* : INT;
Scope_T_DK_Steigband2:REAL;
Scope_T_DK_Steigband2_Visu:REAL;
Scope_T_DK_Steigband3_IN AT%I* : INT;
Scope_T_DK_Steigband3:REAL;
Scope_T_DK_Steigband3_Visu:REAL;
Scope_T_DK_Steigband4_IN AT%I* : INT;
Scope_T_DK_Steigband4:REAL;
Scope_T_DK_Steigband4_Visu:REAL;
Scope_Temp_Heatmatt1_IN  AT%I* : INT;
Scope_Temp_Heatmatt2_IN  AT%I* : INT;
Scope_Temp_Heatmatt3_IN  AT%I* : INT;
Scope_Temp_Heatmatt4_IN  AT%I* : INT;
Scope_Temp_Heatmatt5_IN  AT%I* : INT;
Scope_Temp_Heatmatt6_IN  AT%I* : INT;
Scope_Temp_Heatmatt7_IN  AT%I* : INT;
Scope_Temp_Heatmatt8_IN  AT%I* : INT;
Scope_Temp_Heatmatt9_IN  AT%I* : INT;
Scope_Temp_Heatmatt10_IN  AT%I* : INT;
Scope_Temp_Heatmatt1 : INT;
Scope_Temp_Heatmatt2 : INT;
Scope_Temp_Heatmatt3 : INT;
Scope_Temp_Heatmatt4 : INT;
Scope_Temp_Heatmatt5 : INT;
Scope_Temp_Heatmatt6 : INT;
Scope_Temp_Heatmatt7 : INT;
Scope_Temp_Heatmatt8 : INT;
Scope_Temp_Heatmatt9 : INT;
Scope_Temp_Heatmatt10 : INT;
Scope_Temp_compressor_Self : INT;
Scope_P_Vor_WT_IN AT%I* : INT;
Scope_P_Vor_WT:REAL;
Scope_P_Vor_WT_Visu:REAL;
Scope_P_Durchfluss_IN AT%I* : INT;
Scope_P_Durchfluss:REAL;
Scope_P_Durchfluss_Visu:REAL;
Scope_P_Komp_Einlass_IN AT%I* : INT;
Scope_P_Komp_Einlass:REAL;
Scope_P_Komp_Einlass_Visu:REAL;
Scope_P_Komp_Auslass_IN AT%I* : INT;
Scope_P_Komp_Auslass:REAL;
Scope_P_Komp_Auslass_Visu:REAL;
Scope_W_Kond_Wasser_IN AT%I* : INT;
Scope_W_Kond_Wasser:REAL;
Scope_W_Kond_Wasser_Visu:REAL;
Scope_O2_IN AT%I* : INT;
Scope_O2:REAL;
Scope_O2_Visu:REAL;



END_VAR

// ---- Global Variables/TwinCAT_Configuration.TcGVL
{attribute 'Tc2GvlVarNames'}
(* Generated automatically by TwinCAT - (read only) *)
VAR_CONFIG
	.Main_Relais AT %QX6.0 : BOOL;	(*  ~ {LinkedWith:TIID^Gerät 4 (RT-Ethernet)^Box 1 (BK9000 192.168.100.5)^Klemme 24 (KL2012)^Kanal 2^Ausgang} *)
	.Feedback_Mainswitch AT %IX154.0 : BOOL;	(*  ~ {LinkedWith:TIID^Gerät 4 (RT-Ethernet)^Box 1 (BK9000 192.168.100.5)^Klemme 19 (KL1104)^Kanal 1^Eingang} *)
	.OUT_Mainswitch AT %QX6.1 : BOOL;	(*  ~ {LinkedWith:TIID^Gerät 4 (RT-Ethernet)^Box 1 (BK9000 192.168.100.5)^Klemme 24 (KL2012)^Kanal 1^Ausgang} *)
	.VDC_24_OK AT %IX154.1 : BOOL;	(*  ~ {LinkedWith:TIID^Gerät 4 (RT-Ethernet)^Box 1 (BK9000 192.168.100.5)^Klemme 19 (KL1104)^Kanal 2^Eingang} *)
	.Sollwert_OUT_NV AT %QB20 : INT;
	.Istwert_IN_NV AT %IB176 : INT;
	.Temp_Heatmatt1_IN AT %IB48 : INT;	(*  ~ {LinkedWith:TIID^Gerät 5 (EtherCAT)^Sensorbox_eingänge^Klemme 24 (EL3314)^TC Inputs Channel 1^Value} *)
	.Temp_Heatmatt2_IN AT %IB50 : INT;	(*  ~ {LinkedWith:TIID^Gerät 5 (EtherCAT)^Sensorbox_eingänge^Klemme 24 (EL3314)^TC Inputs Channel 3^Value} *)
	.Temp_Heatmatt3_IN AT %IB52 : INT;	(*  ~ {LinkedWith:TIID^Gerät 5 (EtherCAT)^Sensorbox_eingänge^Klemme 25 (EL3314)^TC Inputs Channel 2^Value} *)
	.Temp_Heatmatt4_IN AT %IB54 : INT;	(*  ~ {LinkedWith:TIID^Gerät 5 (EtherCAT)^Sensorbox_eingänge^Klemme 25 (EL3314)^TC Inputs Channel 4^Value} *)
	.Temp_Heatmatt5_IN AT %IB56 : INT;	(*  ~ {LinkedWith:TIID^Gerät 5 (EtherCAT)^Sensorbox_eingänge^Klemme 25 (EL3314)^TC Inputs Channel 3^Value} *)
	.Temp_Heatmatt6_IN AT %IB58 : INT;	(*  ~ {LinkedWith:TIID^Gerät 5 (EtherCAT)^Sensorbox_eingänge^Klemme 25 (EL3314)^TC Inputs Channel 1^Value} *)
	.Temp_Heatmatt7_IN AT %IB60 : INT;	(*  ~ {LinkedWith:TIID^Gerät 5 (EtherCAT)^Sensorbox_eingänge^Klemme 24 (EL3314)^TC Inputs Channel 2^Value} *)
	.Temp_Heatmatt8_IN AT %IB62 : INT;	(*  ~ {LinkedWith:TIID^Gerät 5 (EtherCAT)^Sensorbox_eingänge^Klemme 24 (EL3314)^TC Inputs Channel 4^Value} *)
	.Temp_Heatmatt9_IN AT %IB64 : INT;	(*  ~ {LinkedWith:TIID^Gerät 5 (EtherCAT)^Sensorbox_eingänge^Klemme 26 (EL3314)^TC Inputs Channel 1^Value} *)
	.Temp_Heatmatt10_IN AT %IB66 : INT;	(*  ~ {LinkedWith:TIID^Gerät 5 (EtherCAT)^Sensorbox_eingänge^Klemme 26 (EL3314)^TC Inputs Channel 2^Value} *)
	.Current_IN_HEAT_Reg_1 AT %IB74 : INT;	(*  ~ {LinkedWith:TIID^Gerät 4 (RT-Ethernet)^Box 1 (BK9000 192.168.100.5)^Klemme 31 (KL3054)^Kanal 2^Daten Ein} *)
	.Current_IN_HEAT_Reg_2 AT %IB76 : INT;	(*  ~ {LinkedWith:TIID^Gerät 4 (RT-Ethernet)^Box 1 (BK9000 192.168.100.5)^Klemme 31 (KL3054)^Kanal 3^Daten Ein} *)
	.Current_IN_HEAT_Reg_3 AT %IB78 : INT;	(*  ~ {LinkedWith:TIID^Gerät 4 (RT-Ethernet)^Box 1 (BK9000 192.168.100.5)^Klemme 31 (KL3054)^Kanal 4^Daten Ein} *)
	.Current_IN_HEAT_Reg_4 AT %IB80 : INT;
	.Current_IN_Compressor_L1 AT %IB82 : INT;	(*  ~ {LinkedWith:TIID^Gerät 4 (RT-Ethernet)^Box 1 (BK9000 192.168.100.5)^Klemme 28 (KL3022)^Kanal 1^Daten Ein} *)
	.Current_IN_Compressor_L2 AT %IB84 : INT;	(*  ~ {LinkedWith:TIID^Gerät 4 (RT-Ethernet)^Box 1 (BK9000 192.168.100.5)^Klemme 28 (KL3022)^Kanal 2^Daten Ein} *)
	.Current_IN_Compressor_L3 AT %IB86 : INT;	(*  ~ {LinkedWith:TIID^Gerät 4 (RT-Ethernet)^Box 1 (BK9000 192.168.100.5)^Klemme 29 (KL3022)^Kanal 1^Daten Ein} *)
	.Current_IN_SteamFan_L1 AT %IB88 : INT;	(*  ~ {LinkedWith:TIID^Gerät 4 (RT-Ethernet)^Box 1 (BK9000 192.168.100.5)^Klemme 30 (KL3054)^Kanal 3^Daten Ein} *)
	.Current_IN_SteamFan_L2 AT %IB90 : INT;	(*  ~ {LinkedWith:TIID^Gerät 4 (RT-Ethernet)^Box 1 (BK9000 192.168.100.5)^Klemme 30 (KL3054)^Kanal 4^Daten Ein} *)
	.Current_IN_SteamFan_L3 AT %IB92 : INT;	(*  ~ {LinkedWith:TIID^Gerät 4 (RT-Ethernet)^Box 1 (BK9000 192.168.100.5)^Klemme 31 (KL3054)^Kanal 1^Daten Ein} *)
	.Current_IN_Fan_L1 AT %IB94 : INT;
	.Current_IN_Fan_L2 AT %IB96 : INT;
	.Current_IN_Fan_L3 AT %IB98 : INT;
	.Current_IN_Complete_L1 AT %IB100 : INT;	(*  ~ {LinkedWith:TIID^Gerät 4 (RT-Ethernet)^Box 1 (BK9000 192.168.100.5)^Klemme 26 (KL3022)^Kanal 2^Daten Ein} *)
	.Current_IN_Complete_L2 AT %IB102 : INT;	(*  ~ {LinkedWith:TIID^Gerät 4 (RT-Ethernet)^Box 1 (BK9000 192.168.100.5)^Klemme 27 (KL3022)^Kanal 1^Daten Ein} *)
	.Current_IN_Complete_L3 AT %IB104 : INT;	(*  ~ {LinkedWith:TIID^Gerät 4 (RT-Ethernet)^Box 1 (BK9000 192.168.100.5)^Klemme 27 (KL3022)^Kanal 2^Daten Ein} *)
	.Compressor_ON AT %QX6.2 : BOOL;	(*  ~ {LinkedWith:TIID^Gerät 4 (RT-Ethernet)^Box 1 (BK9000 192.168.100.5)^Klemme 23 (KL2012)^Kanal 1^Ausgang} *)
	.Compressor_Switch_ON AT %QX6.3 : BOOL;	(*  ~ {LinkedWith:TIID^Gerät 4 (RT-Ethernet)^Box 1 (BK9000 192.168.100.5)^Klemme 21 (KL2114)^Kanal 1^Ausgang} *)
	.Compressor_OK AT %IX154.2 : BOOL;	(*  ~ {LinkedWith:TIID^Gerät 4 (RT-Ethernet)^Box 1 (BK9000 192.168.100.5)^Klemme 20 (KL1104)^Kanal 2^Eingang} *)
	.Compressor_Circuit_breaker AT %IX154.3 : BOOL;	(*  ~ {LinkedWith:TIID^Gerät 4 (RT-Ethernet)^Box 1 (BK9000 192.168.100.5)^Klemme 20 (KL1104)^Kanal 1^Eingang} *)
	.Compressor_Setpoint_OUT AT %QB0 : INT;	(*  ~ {LinkedWith:TIID^Gerät 4 (RT-Ethernet)^Box 1 (BK9000 192.168.100.5)^Klemme 32 (KL4002)^Kanal 1^Daten Aus} *)
	.Compressor_Actual_Turn_IN AT %IB144 : INT;	(*  ~ {LinkedWith:TIID^Gerät 4 (RT-Ethernet)^Box 1 (BK9000 192.168.100.5)^Klemme 25 (KL3022)^Kanal 1^Daten Ein} *)
	.Compressor_PT100_value AT %IB146 : INT;	(*  ~ {LinkedWith:TIID^Gerät 5 (EtherCAT)^Heizbox^Klemme 10 (EL3214)^RTD Inputs Channel 1^Value} *)
	.Compressor_PT100_error AT %IX154.4 : BOOL;	(*  ~ {LinkedWith:TIID^Gerät 5 (EtherCAT)^Heizbox^Klemme 10 (EL3214)^RTD Inputs Channel 1^Status^Error} *)
	.Fan_ON AT %QX32.0 : BOOL;	(*  ~ {LinkedWith:TIID^Gerät 4 (RT-Ethernet)^Box 1 (BK9000 192.168.100.5)^Klemme 21 (KL2114)^Kanal 4^Ausgang} *)
	.Fan_OK AT %IX154.5 : BOOL;	(*  ~ {LinkedWith:TIID^Gerät 4 (RT-Ethernet)^Box 1 (BK9000 192.168.100.5)^Klemme 20 (KL1104)^Kanal 3^Eingang} *)
	.Setpoint_Fan_OUT AT %QB2 : INT;	(*  ~ {LinkedWith:TIID^Gerät 4 (RT-Ethernet)^Box 1 (BK9000 192.168.100.5)^Klemme 32 (KL4002)^Kanal 2^Daten Aus} *)
	.Fan_Actual_Turn_IN AT %IB148 : INT;	(*  ~ {LinkedWith:TIID^Gerät 4 (RT-Ethernet)^Box 1 (BK9000 192.168.100.5)^Klemme 25 (KL3022)^Kanal 2^Daten Ein} *)
	.FAN_Switch_ON AT %QX6.5 : BOOL;	(*  ~ {LinkedWith:TIID^Gerät 4 (RT-Ethernet)^Box 1 (BK9000 192.168.100.5)^Klemme 21 (KL2114)^Kanal 2^Ausgang} *)
	.SteamFan_ON AT %QX6.6 : BOOL;	(*  ~ {LinkedWith:TIID^Gerät 4 (RT-Ethernet)^Box 1 (BK9000 192.168.100.5)^Klemme 22 (KL2114)^Kanal 3^Ausgang} *)
	.Setpoint_SteamFan_OUT AT %QB4 : INT;	(*  ~ {LinkedWith:TIID^Gerät 4 (RT-Ethernet)^Box 1 (BK9000 192.168.100.5)^Klemme 33 (KL4002)^Kanal 1^Daten Aus} *)
	.SteamFan_Actual_Turn_IN AT %IB150 : INT;	(*  ~ {LinkedWith:TIID^Gerät 4 (RT-Ethernet)^Box 1 (BK9000 192.168.100.5)^Klemme 26 (KL3022)^Kanal 1^Daten Ein} *)
	.SteamFAN_Switch_ON AT %QX6.7 : BOOL;	(*  ~ {LinkedWith:TIID^Gerät 4 (RT-Ethernet)^Box 1 (BK9000 192.168.100.5)^Klemme 21 (KL2114)^Kanal 3^Ausgang} *)
	.SteamFan_PTC_IN AT %IX154.7 : BOOL;	(*  ~ {LinkedWith:TIID^Gerät 5 (EtherCAT)^Klemme 41 (EK1200)^Klemme 3 (EL1382)^Channel 1^Input} *)
	.SteamFan_PTC_Error AT %IX155.0 : BOOL;	(*  ~ {LinkedWith:TIID^Gerät 5 (EtherCAT)^Klemme 41 (EK1200)^Klemme 3 (EL1382)^Channel 1^Error} *)
	.Heizelement_Auffangbecken_Mainswitch AT %QX8.4 : BOOL;	(*  ~ {LinkedWith:TIID^Gerät 4 (RT-Ethernet)^Box 1 (BK9000 192.168.100.5)^Klemme 22 (KL2114)^Kanal 1^Ausgang} *)
	.Heat_matt1 AT %QX9.0 : BOOL;	(*  ~ {LinkedWith:TIID^Gerät 5 (EtherCAT)^Sensorbox_Relais^Box 54 (BK1250)^Klemme 7 (KL2631)^Kanal 1^Ausgang} *)
	.Heat_matt2 AT %QX9.1 : BOOL;	(*  ~ {LinkedWith:TIID^Gerät 5 (EtherCAT)^Sensorbox_Relais^Box 54 (BK1250)^Klemme 8 (KL2631)^Kanal 1^Ausgang} *)
	.Heat_matt3 AT %QX9.2 : BOOL;	(*  ~ {LinkedWith:TIID^Gerät 5 (EtherCAT)^Sensorbox_Relais^Box 54 (BK1250)^Klemme 9 (KL2631)^Kanal 1^Ausgang} *)
	.Heat_matt4 AT %QX9.3 : BOOL;	(*  ~ {LinkedWith:TIID^Gerät 5 (EtherCAT)^Sensorbox_Relais^Box 54 (BK1250)^Klemme 10 (KL2631)^Kanal 1^Ausgang} *)
	.Heat_matt5 AT %QX9.4 : BOOL;	(*  ~ {LinkedWith:TIID^Gerät 5 (EtherCAT)^Sensorbox_Relais^Box 54 (BK1250)^Klemme 12 (KL2631)^Kanal 1^Ausgang} *)
	.Heat_matt6 AT %QX9.5 : BOOL;	(*  ~ {LinkedWith:TIID^Gerät 5 (EtherCAT)^Sensorbox_Relais^Box 54 (BK1250)^Klemme 13 (KL2631)^Kanal 1^Ausgang} *)
	.Heat_matt7 AT %QX9.6 : BOOL;	(*  ~ {LinkedWith:TIID^Gerät 5 (EtherCAT)^Sensorbox_Relais^Box 54 (BK1250)^Klemme 14 (KL2631)^Kanal 1^Ausgang} *)
	.Heat_matt8 AT %QX9.7 : BOOL;	(*  ~ {LinkedWith:TIID^Gerät 5 (EtherCAT)^Sensorbox_Relais^Box 54 (BK1250)^Klemme 15 (KL2631)^Kanal 1^Ausgang} *)
	.Heat_matt9 AT %QX10.0 : BOOL;	(*  ~ {LinkedWith:TIID^Gerät 5 (EtherCAT)^Sensorbox_eingänge^Klemme 18 (EL2828)^Channel 6^Output} *)
	.Heat_matt10 AT %QX10.1 : BOOL;	(*  ~ {LinkedWith:TIID^Gerät 5 (EtherCAT)^Sensorbox_eingänge^Klemme 18 (EL2828)^Channel 7^Output} *)
	.HEAT_Reg_Mainswitch_OUT AT %QX10.6 : BOOL;	(*  ~ {LinkedWith:TIID^Gerät 4 (RT-Ethernet)^Box 1 (BK9000 192.168.100.5)^Klemme 22 (KL2114)^Kanal 2^Ausgang} *)
	.HEAT_Reg_1_OUT AT %QX10.2 : BOOL;	(*  ~ {LinkedWith:TIID^Gerät 5 (EtherCAT)^Heizbox^Klemme 7 (EL2828)^Channel 1^Output} *)
	.HEAT_Reg_2_OUT AT %QX10.3 : BOOL;	(*  ~ {LinkedWith:TIID^Gerät 5 (EtherCAT)^Heizbox^Klemme 7 (EL2828)^Channel 2^Output} *)
	.HEAT_Reg_3_OUT AT %QX10.4 : BOOL;	(*  ~ {LinkedWith:TIID^Gerät 5 (EtherCAT)^Heizbox^Klemme 7 (EL2828)^Channel 7^Output} *)
	.HEAT_Reg_4_OUT AT %QX10.5 : BOOL;	(*  ~ {LinkedWith:TIID^Gerät 5 (EtherCAT)^Heizbox^Klemme 7 (EL2828)^Channel 8^Output} *)
	.Heat_matt_Group1_1_4_manu AT %QX12.0 : BOOL;	(*  ~ {LinkedWith:TIID^Gerät 5 (EtherCAT)^Sensorbox_eingänge^Klemme 18 (EL2828)^Channel 1^Output} *)
	.Heat_matt_Group2_5_8_manu AT %QX12.1 : BOOL;	(*  ~ {LinkedWith:TIID^Gerät 5 (EtherCAT)^Sensorbox_eingänge^Klemme 18 (EL2828)^Channel 2^Output} *)
	.Heat_matt_Group3_9_10_manu AT %QX12.2 : BOOL;	(*  ~ {LinkedWith:TIID^Gerät 5 (EtherCAT)^Sensorbox_eingänge^Klemme 18 (EL2828)^Channel 3^Output} *)
	.LED_RED_OUT AT %QX11.1 : BOOL;	(*  ~ {LinkedWith:TIID^Gerät 5 (EtherCAT)^Sensorbox_eingänge^Klemme 19 (EL2828)^Channel 3^Output} *)
	.LED_green_OUT AT %QX11.2 : BOOL;	(*  ~ {LinkedWith:TIID^Gerät 5 (EtherCAT)^Sensorbox_eingänge^Klemme 19 (EL2828)^Channel 1^Output} *)
	.LED_yellow_OUT AT %QX11.3 : BOOL;	(*  ~ {LinkedWith:TIID^Gerät 5 (EtherCAT)^Sensorbox_eingänge^Klemme 19 (EL2828)^Channel 2^Output} *)
	.LED_white_OUT AT %QX11.4 : BOOL;	(*  ~ {LinkedWith:TIID^Gerät 5 (EtherCAT)^Sensorbox_eingänge^Klemme 19 (EL2828)^Channel 4^Output} *)
END_VAR

// ---- Global Variables/Variablen_Konfiguration.TcGVL
{attribute 'Tc2GvlVarNames'}
VAR_CONFIG
END_VAR

// ---- POUs/SCL_MAIN.TcPOU
PROGRAM SCL_MAIN
VAR

	(*Funktionsaufrufe*)


	Puls_GEN_Watervalve:FB_Blink;

	



	Average1:Average;
	Average2:Average;
	Average3:Average;
	Average4:Average;
	Average5:Average;
	Average6:Average;
	Average7:Average;
	Average8:Average;
	Average9:Average;
	Average10:Average;
	Average11:Average;
	Average12:Average;
	Average13:Average;
	Average14:Average;
	Average15:Average;
	Average16:Average;
	Average17:Average;
	Average18:Average;
	Average19:Average;
	Average20:Average;
	Average21:Average;
	Average22:Average;
	Average23:Average;


	F_TRIG1:F_TRIG;
	R_TRIG1:R_TRIG;

	OUT_FTRIG1:BOOL;
	C_NOT_AUS: INT;




	(*Rückstellung der Ventilsequenz vom Manuelltaster der einzelnen Ventile*)
	F_TRIG2:F_TRIG;
	F_TRIG3:F_TRIG;
	F_TRIG4:F_TRIG;
	F_TRIG5:F_TRIG;
	F_TRIG6:F_TRIG;
	F_TRIG7:F_TRIG;
	F_TRIG8:F_TRIG;
	F_TRIG9:F_TRIG;
	F_TRIG10:F_TRIG;
	F_TRIG11:F_TRIG;
	F_TRIG12:F_TRIG;


	F_TRIG20:F_TRIG;


	R_TRIG10:R_TRIG;
	R_TRIG11:R_TRIG;
	R_TRIG12:R_TRIG;
	R_TRIG13:R_TRIG;




	SR1:SR;
	SR2:SR;
	SR3:SR;
	SR4:SR;
	SR5:SR;
	SR6:SR;
	SR7:SR;
	SR8:SR;
	SR9:SR;
	SR10:SR;
	SR11:SR;
	SR12:SR;
	SR13:SR;





	Start_Programm: BOOL;
	Res_Start_Programm: BOOL;
	Set_Start_Programm: BOOL;
	Emergency: BOOL;
	nCounter : UINT;




	(*ZEITEN*)

	TON1:TP;
	IN_T1:BOOL;
	OUT_T1:BOOL;
	TON2:TON;
	IN_T2:BOOL;
	OUT_T2:BOOL;
	TON3:TON;
	IN_T3:BOOL;
	OUT_T3:BOOL;
	ET_T3:TIME;
	TON4:TON;
	IN_T4:BOOL;
	OUT_T4:BOOL;
	TON5:TON;
	IN_T5:BOOL;
	OUT_T5:BOOL;
	TON6:TON;
	IN_T6:BOOL;
	OUT_T6:BOOL;
	TON7:TON;
	IN_T7:BOOL;
	OUT_T7:BOOL;
	TON8:TON;
	IN_T8:BOOL;
	OUT_T8:BOOL;
	TON9:TON;
	IN_T9:BOOL;
	OUT_T9:BOOL;
	TON10:TON;
	IN_T10:BOOL;
	OUT_T10:BOOL;
	TON11:TON;
	IN_T11:BOOL;
	OUT_T11:BOOL;
	TON12:TON;
	IN_T12:BOOL;
	OUT_T12:BOOL;
	TON13:TON;
	IN_T13:BOOL;
	OUT_T13:BOOL;
	TON14:TON;
	IN_T14:BOOL;
	OUT_T14:BOOL;
	TON15:TON;
	IN_T15:BOOL;
	OUT_T15:BOOL;
	TON16:TON;
	IN_T16:BOOL;
	OUT_T16:BOOL;
	TON17:TON;
	IN_T17:BOOL;
	OUT_T17:BOOL;
	TON18:TON;
	IN_T18:BOOL;
	OUT_T18:BOOL;
	TON19:TON;
	IN_T19:BOOL;
	OUT_T19:BOOL;
	TON20:TON;
	IN_T20:BOOL;
	OUT_T20:BOOL;
	TON21:TON;
	IN_T21:BOOL;
	OUT_T21:BOOL;
	TON22:TON;
	IN_T22:BOOL;
	OUT_T22:BOOL;
	TON23:TON;
	IN_T23:BOOL;
	OUT_T23:BOOL;
	TON24:TON;
	IN_T24:BOOL;
	OUT_T24:BOOL;
	TON25:TON;
	IN_T25:BOOL;
	OUT_T25:BOOL;
	TON26:TON;
	IN_T26:BOOL;
	OUT_T26:BOOL;

	TP30:TP;
	IN_T30:BOOL;
	OUT_T30:BOOL;













	Ton_Pulsgen:TP;
	OUT_Pulsgen: BOOL;

	(*Hyterese DES*)


	TON100:TON;
	IN_T100:BOOL;
	OUT_T100:BOOL;
	TON101:TON;
	IN_T101:BOOL;
	OUT_T101:BOOL;
	TON102:TON;
	IN_T102:BOOL;
	OUT_T102:BOOL;
	TON103:TON;
	IN_T103:BOOL;
	OUT_T103:BOOL;
	TON104:TON;
	IN_T104:BOOL;
	OUT_T104:BOOL;
	TON105:TON;
	IN_T105:BOOL;
	OUT_T105:BOOL;
	TON106:TON;
	IN_T106:BOOL;
	OUT_T106:BOOL;
	TON107:TON;
	IN_T107:BOOL;
	OUT_T107:BOOL;


	TON108:TON;
	IN_T108:BOOL;
	OUT_T108:BOOL;


	Hyst1:Meine_HYST;
	Hyst2:Meine_HYST;
	Hyst3:Meine_HYST;
	Hyst4:Meine_Hyst;
	Hyst5:Meine_Hyst;
	Hyst6:Meine_Hyst;
	Hyst7:Meine_Hyst;
	Hyst8:Meine_Hyst;
	Hyst9:Meine_HYST;
	Hyst10:Meine_HYST;


	Change_dir: BOOL;

	CTU1:CTU;
	Res_C1: BOOL;
	C_up1:BOOL;
	(*C_val1: WORD; IST Global*)

	CTU2:CTU;
	Res_C2: BOOL;
	C_up2:BOOL;
	C_val2: WORD;

	CTU3:CTU;
	Res_C3: BOOL;
	C_up3:BOOL;
	C_val3: WORD;

	CTU4:CTU;
	Res_C4: BOOL;
	C_up4:BOOL;
	C_val4: WORD;

	bBlink:BOOL;
	bStart:BOOL;
	C_Diff: INT;
	C_Valve_Seq_Prop: INT;

	Start_Auto_Export_INT: INT;
	PWM: BOOL;
	fbWriteRegs 	:	 FB_MBWriteRegs;


	Current_OUT_Complete_L1_temp: REAL;
	Current_OUT_Complete_L2_temp: REAL;
	Current_OUT_Complete_L3_temp: REAL;
	C_test: INT;
	bError:BOOL;

	FAN_Switch_ON_Manu: BOOL;
	
	
	
	
	PID_Test: FB_BasicPID;
	fSetpointValue_IN: LREAL;
	fActualValue_IN: LREAL;
	bReset_IN: BOOL;
	fCtrlOutput_OUT: LREAL;
	
	
	
	Controller:Controller;
	
	
	
	
	
	
	//Für UDP Kommunikation:
	
	bSendOnceToItself	: BOOL;(* Rising edge at this variable sends message to local host/port (itself) *)
	bSendOnceToRemote	: BOOL;(* Rising edge at this variable sends message to the remote host/port *)
	sSrvNetId			: T_AmsNetID 	:= '';(* TwinCAT TCP/IP server network address. Default: empty string. *)
	sLocalHost			: T_IPv4Addr 	:= '192.168.100.88';(* Local address: String containing an (Ipv4) Internet Protocol dotted address. *)
	nLocalPort			: UDINT			:= 1001;(* Local address: IP port number. *)
	sRemoteHost			: T_IPv4Addr 	:= '192.168.100.101';(* Remote address: String containing an (Ipv4) Internet Protocol dotted address. *)
	nRemotePort			: UDINT 		:= 1000;(* Remote address: IP port number. *)
	bEnable				: BOOL 			:= TRUE;(* TRUE => Enable/connect, FALSE => Disable/disconnect *)
	bLog				: BOOL			:= TRUE;(* TRUE => Enable log message output, FALSE => Disable *)

	fbPeerToPeer		: FB_PeerToPeer := ( sPrefix := 'PeerToPeerA::' ); //für ehemals test mit IAS
	
   	fbTx				: FB_FrameFifo;
   	fbRx				: FB_FrameFifo;
   	fbLog				: FB_LogFifo;
	
   	stSendTo			: ST_FrameFifoEntry;
   	stReceivedFrom		: ST_FrameFifoEntry;
	sLoggedMessage		: T_MaxString;

   	fbCloseAll 			: FB_SocketCloseAll;
   	bInitialize			: BOOL := TRUE;
	nErrID_FBClose		:UDINT;

END_VAR




VAR_INPUT



END_VAR
VAR_IN_OUT

END_VAR



(* ______________________Version3
Erstelldatum:	März.02020
Ersteller:	Daniel Meyer
Zweck:	Grundlageprogramm Aquaero Triss (Anlage3) *)

(*Funktionsaufrufe*)
(*Controller_functions();*)
(*Startbedingungen des  Monstrators*)













Istwert_IN_NV_OUT:=(Istwert_IN_NV*100)/32767;



(*_______________________________________________________________________________Skallierungen________________________________________________________________________*)




(*_________________________________Dieser Ventilator brauchts zurzeit nicht mehr
(*Ventilator*)

Setpoint_Fan_OUT:=(Setpoint_Fan_IN*32767)/100;

(*Wichtig!!! Zurzeit ist dies die Leistungsabgabe  20mA = 100% = 32767= 2.2KW*)

Fan_Actual_Turn:=(Fan_Actual_Turn_IN*100.0)/32767;	(*0-100% Aufgrund von tests mit der Solldrehzahl*)
*)



(*Umdampfventilatorr*)

Setpoint_SteamFan_OUT:=(Setpoint_SteamFan_IN*32767)/100;

SteamFan_Actual_Turn:=(SteamFan_Actual_Turn_IN*2870)/32767;

IF SteamFAN_Switch_ON_manu THEN SteamFan_OK:=TRUE; ELSE SteamFan_OK:=FALSE;	END_IF;



(*Kompressoren*)

Compressor_Setpoint_OUT:=(Setpoint_Compressor_IN*16384)/100;	(*Zurzeit ist beim Kompressor bei 5V der Max. Frequenzausgang.!! Noch kontrollieren warum??*)



(*Wichtig!!! Zurzeit ist dies die Leistungsabgabe 20mA = 200% von max Leistung = 6KW*)

Compressor_Actual_Turn:=(Compressor_Actual_Turn_IN*100.0)/4444;	(*0-100% Aufgrund von tests mit der Solldrehzahl*)

(*0-100%*)








(*Steig & Normalförderer*)

Setpoint_M_Belt_Feeder_OUT:=(Setpoint_M_Belt_Feeder_IN*16384)/100;	(*Zurzeit ist beim Schneider Electric -FU bei 5V der Max. Frequenzausgang.!! Noch kontrollieren warum??*)

M_Belt_Feeder_Actual_Turn:=(M_Belt_Feeder_Actual_Turn_IN*32767)/100;




Setpoint_M_Belts_OUT:=(Setpoint_M_Belts_IN*32767)/100;

M_Belts_Actual_Turn:=(M_Belts_Actual_Turn_IN*100.0)/32767;	(*0-100% *)










(*_____Strom und Energie_____*)


(*zumteil auch: *50.0)/16383.5) bei 5VDC!!!*)

(*
Average1(Input_AV:=((Current_IN_HZE_Auffangbecken_L1*50.0)/16384) , OUTPUT_AV=>Current_OUT_SteamVenti_L1);(*Wichtig!! die Messung wird zurzeit ueber einen 0bis10v Spannungseingang gelesen*)
Average2(Input_AV:=((Current_IN_HZE_Auffangbecken_L2*50.0)/32767.0) , OUTPUT_AV=>Current_OUT_SteamVenti_L2);
Average3(Input_AV:=((Current_IN_HZE_Auffangbecken_L3*50.0)/32767.0) , OUTPUT_AV=>Current_OUT_SteamVenti_L3);
*)


Average4(Input_AV:=((Current_IN_HEAT_Reg_1*10.0)/32767.0) , OUTPUT_AV=>Current_OUT_HEAT_Reg_1);
Average5(Input_AV:=((Current_IN_HEAT_Reg_2*10.0)/32767.0) , OUTPUT_AV=>Current_OUT_HEAT_Reg_2);
Average6(Input_AV:=((Current_IN_HEAT_Reg_3*10.0)/32767.0) , OUTPUT_AV=>Current_OUT_HEAT_Reg_3);
Average7(Input_AV:=((Current_IN_HEAT_Reg_4*10.0)/32767.0) , OUTPUT_AV=>Current_OUT_HEAT_Reg_4);

Average20(Input_AV:=((Current_IN_HEAT_Reg_5*10.0)/32767.0) , OUTPUT_AV=>Current_OUT_HEAT_Reg_5);
Average21(Input_AV:=((Current_IN_HEAT_Reg_6*10.0)/32767.0) , OUTPUT_AV=>Current_OUT_HEAT_Reg_6);
Average22(Input_AV:=((Current_IN_HEAT_Reg_7*10.0)/32767.0) , OUTPUT_AV=>Current_OUT_HEAT_Reg_7);
Average23(Input_AV:=((Current_IN_HEAT_Reg_8*10.0)/32767.0) , OUTPUT_AV=>Current_OUT_HEAT_Reg_8);




Average8(Input_AV:=((Current_IN_Compressor_L1*10.0)/32767.0) , OUTPUT_AV=>Current_OUT_Compressor_L1);
Average9(Input_AV:=((Current_IN_Compressor_L2*10.0)/32767.0) , OUTPUT_AV=>Current_OUT_Compressor_L2);
Average10(Input_AV:=((Current_IN_Compressor_L3*10.0)/32767.0) , OUTPUT_AV=>Current_OUT_Compressor_L3);

Average11(Input_AV:=((Current_IN_SteamFan_L1*10.0)/32767.0) , OUTPUT_AV=>Current_OUT_AdsorbtionsVenti_L1);(*Wichtig!! Ist zurzeit Adsobrtionslüfter!!!*)
Average12(Input_AV:=((Current_IN_SteamFan_L2*10.0)/32767.0) , OUTPUT_AV=>Current_OUT_AdsorbtionsVenti_L2);(*Wichtig!! Ist zurzeit Adsobrtionslüfter!!!*)
Average13(Input_AV:=((Current_IN_SteamFan_L3*10.0)/32767.0) , OUTPUT_AV=>Current_OUT_AdsorbtionsVenti_L3);(*Wichtig!! Ist zurzeit Adsobrtionslüfter!!!*)

Average14(Input_AV:=((Current_IN_Fan_L1*10.0)/32767.0) , OUTPUT_AV=>Current_OUT_Fan_L1);
Average15(Input_AV:=((Current_IN_Fan_L2*10.0)/32767.0) , OUTPUT_AV=>Current_OUT_Fan_L2);
Average16(Input_AV:=((Current_IN_Fan_L3*10.0)/32767.0) , OUTPUT_AV=>Current_OUT_Fan_L3);

Average17(Input_AV:=((Current_IN_Complete_L1*20.0)/32767.0) , OUTPUT_AV=>Current_OUT_Complete_L1 );
Average18(Input_AV:=((Current_IN_Complete_L2*20.0)/32767.0) , OUTPUT_AV=>Current_OUT_Complete_L2 );
Average19(Input_AV:=((Current_IN_Complete_L3*20.0)/32767.0) , OUTPUT_AV=>Current_OUT_Complete_L3 );











(*1.732= Wurzel 3, es wird angenommen das Cos PHI = 0 und Wirkungsgrad = 0.8 ist*)

Energy_OUT_HZE_Auffangbecken_L1:=(Current_OUT_SteamVenti_L1*400*1.732*0.8)/1000;
Energy_OUT_HZE_Auffangbecken_L2:=(Current_OUT_SteamVenti_L2*400*1.732*0.8)/1000;
Energy_OUT_HZE_Auffangbecken_L3:=(Current_OUT_SteamVenti_L3*400*1.732*0.8)/1000;
Energy_OUT_HEAT_Reg_1:=(Current_OUT_HEAT_Reg_1*400*1.732*0.8)/1000;
Energy_OUT_HEAT_Reg_2:=(Current_OUT_HEAT_Reg_2*400*1.732*0.8)/1000;
Energy_OUT_HEAT_Reg_3:=(Current_OUT_HEAT_Reg_3*400*1.732*0.8)/1000; 
Energy_OUT_HEAT_Reg_4:=(Current_OUT_HEAT_Reg_4*400*1.732*0.8)/1000;

Energy_OUT_HEAT_Reg_5:=(Current_OUT_HEAT_Reg_5*400*1.732*0.8)/1000;
Energy_OUT_HEAT_Reg_6:=(Current_OUT_HEAT_Reg_6*400*1.732*0.8)/1000;
Energy_OUT_HEAT_Reg_7:=(Current_OUT_HEAT_Reg_7*400*1.732*0.8)/1000;
Energy_OUT_HEAT_Reg_8:=(Current_OUT_HEAT_Reg_8*400*1.732*0.8)/1000;





Energy_OUT_Compressor_L1:=(Current_OUT_Compressor_L1*400*1.732*0.8)/1000;
Energy_OUT_Compressor_L1:=(Current_OUT_Compressor_L1*400*1.732*0.8)/1000;
Energy_OUT_Compressor_L1:=(Current_OUT_Compressor_L1*400*1.732*0.8)/1000;
Energy_OUT_SteamFan_L1:=(Current_OUT_AdsorbtionsVenti_L1*400*1.732*0.8)/1000;
Energy_OUT_SteamFan_L2:=(Current_OUT_AdsorbtionsVenti_L2*400*1.732*0.8)/1000;
Energy_OUT_SteamFan_L3:=(Current_OUT_AdsorbtionsVenti_L3*400*1.732*0.8)/1000;
Energy_OUT_Fan_L1:=(Current_OUT_Fan_L1*400*1.732*0.8)/1000;
Energy_OUT_Fan_L2:=(Current_OUT_Fan_L2*400*1.732*0.8)/1000;
Energy_OUT_Fan_L3:=(Current_OUT_Fan_L3*400*1.732*0.8)/1000;
Energy_OUT_Complete_L1:=(Current_OUT_Complete_L1*400*1.732*0.8)/1000;
Energy_OUT_Complete_L2:=(Current_OUT_Complete_L2*400*1.732*0.8)/1000;
Energy_OUT_Complete_L3:=(Current_OUT_Complete_L3*400*1.732*0.8)/1000;









T_Vor_WT_Visu:=(T_Vor_WT_IN*150)/32767;(*SE-T 1.01*)
T_Nach_WT_Visu:=(T_Nach_WT_IN*150)/32767;(*SE-T 1.02*)

T_HE_Einduesung_Oben_Visu:=T_HE_Einduesung_Oben_IN/10.0;(*SE-T 1.03*)
T_HE_Einduesung_Unten_Visu:=T_HE_Einduesung_Unten_IN/10.0;(*SE-T 1.04*)

T_Einduesung_Oben_Visu:=T_Einduesung_Oben_IN/10.0;(*SE-T 1.05*)
T_Einduesung_Unten_Visu:=T_Einduesung_Unten_IN/10.0;(*SE-T 1.06*)

T_Absaugung_Oben_Visu:=(T_Absaugung_Oben_IN*150.0)/32767;(*SE-T 1.07*)
T_Absaugung_Unten_Visu:=(T_Absaugung_Unten_IN*150.0)/32767;(*SE-T 1.08*)

T_Vor_UmdampfLuefter_Visu:=(T_Vor_UmdampfLuefter_IN*150.0)/32767;(*SE-T 1.09*)


T_Komp_Einlass_Visu:=(T_Komp_Einlass_IN*150.0)/32767;(*SE-T 2.01*)
T_Komp_Auslass_Visu:=(T_Komp_Auslass_IN*150.0)/32767;(*SE-T 2.02*)
T_Kond_Auslass_Visu:=T_Kond_Auslass_IN/10.0;(*SE-T 2.03*)



T_DK_oben_Visu:=T_DK_oben_IN/10.0;(*SE-T 3.01*)
T_DK_mitte_Visu:=T_DK_mitte_IN/10.0;(*SE-T 3.02*)
T_DK_unten_Visu:=T_DK_unten_IN/10.0;(*SE-T 3.03*)


T_Mat_Auslass1_Visu:=T_Mat_Auslass1_IN/10.0;(*SE-T 3.71*)
T_Mat_Auslass2_Visu:=T_Mat_Auslass2_IN/10.0;(*SE-T 3.72*)
T_Mat_Auslass3_Visu:=T_Mat_Auslass3_IN/10.0;(*SE-T 3.73*)
T_Mat_Auslass4_Visu:=T_Mat_Auslass4_IN/10.0;(*SE-T 3.74*)

T_Mat_Auslass5_Visu:=T_Mat_Auslass5_IN/10.0;(*SE-T 3.71*)
T_Mat_Auslass6_Visu:=T_Mat_Auslass6_IN/10.0;(*SE-T 3.72*)
T_Mat_Auslass7_Visu:=T_Mat_Auslass7_IN/10.0;(*SE-T 3.73*)
T_Mat_Auslass8_Visu:=T_Mat_Auslass8_IN/10.0;(*SE-T 3.74*)


T_Komp_Gehaeuse_Visu:=T_Komp_Gehaeuse_IN/10.0; (*SE-T 4.01*)



T_DK_Band_oben1_Visu:=T_DK_Band_oben1_IN/10.0;(*SE-T 1.81*)
T_DK_Band_oben2_Visu:=T_DK_Band_oben2_IN/10.0;(*SE-T  1.82*)
T_DK_Band_oben3_Visu:=T_DK_Band_oben3_IN/10.0;(*SE-T 1.83*)

T_DK_Band_unten1_Visu:=T_DK_Band_unten1_IN/10.0;(*SE-T  1.91*)
T_DK_Band_unten2_Visu:=T_DK_Band_unten2_IN/10.0;(*SE-T 1.92*)
T_DK_Band_unten3_Visu:=T_DK_Band_unten3_IN/10.0;(*SE-T 1.93*)


T_DK_Steigband1_Visu:=T_DK_Steigband1_IN/10.0;(*SE-T 3.81*)
T_DK_Steigband2_Visu:=T_DK_Steigband2_IN/10.0;(*SE-T 3.82*)
T_DK_Steigband3_Visu:=T_DK_Steigband3_IN/10.0;(*SE-T 3.83*)
T_DK_Steigband4_Visu:=T_DK_Steigband4_IN/10.0;(*SE-T 3.84*)



Temp_Heatmatt1:=(Temp_Heatmatt1_IN/10);
Temp_Heatmatt2:=(Temp_Heatmatt2_IN/10);
Temp_Heatmatt3:=(Temp_Heatmatt3_IN/10);
Temp_Heatmatt4:=(Temp_Heatmatt4_IN/10);
Temp_Heatmatt5:=(Temp_Heatmatt5_IN/10);
Temp_Heatmatt6:=(Temp_Heatmatt6_IN/10);
Temp_Heatmatt7:=(Temp_Heatmatt7_IN/10);
Temp_Heatmatt8:=(Temp_Heatmatt8_IN/10);
Temp_Heatmatt9:=(Temp_Heatmatt9_IN/10);
Temp_Heatmatt10:=(Temp_Heatmatt10_IN/10);





P_Komp_Einlass_Visu:=(P_Komp_Einlass_IN*2500)/32767;(*SE-P 2.11 STS 2500bara**)
P_Komp_Auslass_Visu:=(P_Komp_Auslass_IN*2500)/32767;(*SE-P 2.12 STS 2500bara**)

W_Kond_Wasser_Visu:=DINT_TO_REAL((W_Kond_Wasser_IN*50000)/32767);(*SE-W 2.31 50000 = g*)

O2_Visu:=(O2_IN*25.0)/32767;(*SE-O2 1.51    25=%O2*)


P_Vor_WT_Visu:=(P_Vor_WT_IN*2500)/32767;(*SE-P 1.11  STS 2500bara*)
(*P_Durchfluss_Visu:=(P_Durchfluss_IN*xy)/32767;(*SE-P 1.44*)*)












IF PTC_IN = FALSE THEN
Motor_HOT:=TRUE;
ELSE
Motor_HOT:=FALSE;
END_IF;

(*


(*Formeln&Berechnungen*)


Ps_311:=TRUNC(((-0.00002405*( T_Vor_KlauenkolbenKomp* T_Vor_KlauenkolbenKomp))+(0.000950471* T_Vor_KlauenkolbenKomp)+6.1226)*EXP((17.62* T_Vor_KlauenkolbenKomp)/(243.15+ T_Vor_KlauenkolbenKomp)));

Ps_26:=TRUNC(((-0.00002405*( T_Des_nach_WT* T_Des_nach_WT))+(0.000950471* T_Des_nach_WT)+6.1226)*EXPT(2.71828,((17.62* T_Des_nach_WT)/(243.15+ T_Des_nach_WT))));


Ps_28:=TRUNC(((-0.00002405*( T_Des_vor_DecicWheel* T_Des_vor_DecicWheel))+(0.000950471* T_Des_vor_DecicWheel)+6.1226)*EXPT(2.71828,((17.62* T_Des_vor_DecicWheel)/(243.15+ T_Des_vor_DecicWheel))));


Ps_23:=TRUNC(((-0.00002405*( T_Des_nach_V_Umdampf* T_Des_nach_V_Umdampf))+(0.000950471* T_Des_nach_V_Umdampf)+6.1226)*EXPT(2.71828,((17.62* T_Des_nach_V_Umdampf)/(243.15+ T_Des_nach_V_Umdampf))));



RelP_TM:=P_Des_nach_WT/Ps_28;
RelP_WT:=P_Des_nach_WT/P_Dampfleitung_comp;
RelP_Out:=P_Des_nach_WT/Ps_23;

*)



(* ps(T)=(-0.00002405*T^2+0.000950471*T+6.1226)*exp(17.62*T/(243.15+T))/1000;*)








(*_______________________________________Not-Aus-Relais-________________________________________________*)


(*Error summen*)

Main_Relais:=(NOT Switch_OFF_Mainswitch AND Main_Relais   ) OR Start_Mainswitch;

F_TRIG20(CLK:= Switch_OFF_Mainswitch , Q=>Start_Auto_Export );

TP30(IN:=Start_Auto_Export , PT:= t#3S, Q=> Start_Auto_Export_OUT , ET=> );




IF RESET_ERROR_Mainswitch THEN
ERROR_Mainswitch:=FALSE;
Main_Relais:=FALSE;
IN_T1:=FALSE;
IN_T2:=FALSE;
END_IF;

IF  Main_Relais = FALSE  THEN
ERROR_Mainswitch:=FALSE;
C_NOT_AUS:=0;
IN_T1:=FALSE;
IN_T2:=FALSE;
END_IF;

CASE C_NOT_AUS OF

	0:	IN_T1:=FALSE;
		IN_T2:=FALSE;
		Mainswitch_OK:=FALSE;
		C_NOT_AUS:=1;

	1: 	IF  Main_Relais THEN

		IN_T1:=TRUE;
		IN_T2:=TRUE;
		C_NOT_AUS:=2;
		ELSE
		C_NOT_AUS:=1;
		END_IF

	2:
		IN_T1:=FALSE;
		C_NOT_AUS:=3;

	3: 	IF Feedback_Mainswitch AND OUT_T2 THEN

		Mainswitch_OK:=TRUE;
		Switch_Heat_group1:=TRUE;
		Switch_Heat_group2 :=TRUE;
		Switch_Heat_group3 :=TRUE;

		(*ELSE IF Feedback_Mainswitch = FALSE THEN
		Mainswitch_OK:=FALSE;*)
		ELSE IF  Feedback_Mainswitch = FALSE AND OUT_T2  THEN
		C_NOT_AUS:=6;
		END_IF
		END_IF


	(*4:	Mainswitch_OK:=TRUE;*)

	6:	IN_T2:=FALSE;
		ERROR_Mainswitch:=TRUE;


		Mainswitch_OK:=FALSE;
		C_NOT_AUS:=7;	(*Zurzeit fertig*)



	100: C_NOT_AUS:=0;

END_CASE

OUT_Mainswitch:=OUT_T1;






	(*Wenn Not-Aus gedrückt wurde, werden folgende Werte zurückgesetzt*)



	(* NOT-AUS*)


	IF Mainswitch_OK = FALSE THEN

	C_DES:=100;
	C_ADS:=100;


	Setpoint_Fan_Visu:=0;
	Setpoint_Compressor_Visu:=0;
	Setpoint_M_Belt_Feeder_Visu:=0;
	Setpoint_M_Belts_Visu:=0;
	Setpoint_SteamFan_Visu:=0;




	FAN_Switch_ON:=FALSE;
	FAN_ON:=FALSE;
	FAN_Switch_ON_Manu:=FALSE;
	FAN_ON_Manu:=FALSE;

	Compressor_Switch_ON:=FALSE;
	Compressor_ON:=FALSE;
	Compressor_Switch_ON_manu:=FALSE;
	Compressor_ON_manu:=FALSE;

	Compressor_cooling_manu :=FALSE;
	Compressor_cooling_auto :=FALSE;
	Compressor_cooling :=FALSE;

	SteamFAN_Switch_ON:=FALSE;
	SteamFAN_Switch_ON_Manu:=FALSE;
	SteamFan_ON:=FALSE;
	SteamFan_ON_manu:=FALSE;


	M_Belts_ON:=FALSE;
	M_Belts_Switch_ON:=FALSE;
	M_Belts_Switch_ON_Manu:=FALSE;
	M_Belts_ON_Manu:=FALSE;


	M_Belt_Feeder_ON:=FALSE;
	M_Belt_Feeder_Switch_ON:=FALSE;
	M_Belt_Feeder_Switch_ON_Manu:=FALSE;
	M_Belt_Feeder_ON_Manu:=FALSE;




	Control_Manu_active:=FALSE;
	Control_Auto_active:=FALSE;


	ELSE








(*Hier beginnt die eigentliche Programmbearbeitung*)






(*Einschalten von Haupt- und Motorrelais*)

(* zurzeit nicht verwendeT


Main_Relais:=(NOT Reset_M_R AND  Main_Relais AND NOT_AUS) OR Set_M_R;

*)

Cabinet_OK:=VDC_24_OK; (* AND---*)




(* Manu / Auto Umschaltung *)



(*Manu/Automodeumschaltung*)

(*Manu/Automodeumschaltung*)

(*Start_Man:=(NOT Reset_man AND Start_Man) OR Set_Man;*)

(* vom Automodus soll man nicht direkt in den Manu Modus schalten können, zuerst muss man den automodus stoppen*)

Control_Manu_active:=(NOT( Reset_man OR Control_Auto ) AND Control_Manu_active AND Mainswitch_OK) OR Control_Manu;
Control_Auto_active:=(NOT Reset_Auto AND Control_Auto_active AND Mainswitch_OK) OR Control_Auto;



(*_________________________________________________________________________________________CONTROL___Manu____________________________________________*)



IF Control_Manu_active THEN




	(*FAN*)

	Setpoint_Fan_IN:= Setpoint_Fan_Visu;

	FAN_Switch_ON:=FAN_Switch_ON_Manu;
	FAN_ON:=FAN_ON_Manu;




	(* Steig & Horizontalbandförderer*)


	IF Activate_controller_M_Belts THEN
	Setpoint_M_Belts_IN:=REAL_TO_INT(fStellwert_M_Belts);
	ELSE
	Setpoint_M_Belts_IN:=Setpoint_M_Belts_Visu;
	END_IF;

	M_Belts_Switch_ON:=M_Belts_Switch_ON_Manu;
	M_Belts_ON:=M_Belts_ON_Manu;






	IF Activate_controller_M_Belt_Feeder THEN
	Setpoint_M_Belt_Feeder_IN:=REAL_TO_INT(fStellwert_M_Belt_Feeder);
	ELSE
	Setpoint_M_Belt_Feeder_IN:=Setpoint_M_Belt_Feeder_Visu;
	END_IF;

	M_Belt_Feeder_Switch_ON:=M_Belt_Feeder_Switch_ON_Manu;
	M_Belt_Feeder_ON:=M_Belt_Feeder_ON_Manu;







	IF Activate_controller_comp THEN
	Setpoint_Compressor_IN:=REAL_TO_INT(fStellwert_comp);
	ELSE
	Setpoint_Compressor_IN:= Setpoint_Compressor_Visu;
	END_IF

	Compressor_Switch_ON:=Compressor_Switch_ON_Manu;
	Compressor_ON:=Compressor_ON_Manu;



	IF Activate_controller_V_Umdampf  THEN
	Setpoint_SteamFan_IN:=REAL_TO_INT(fStellwert_V_Umdampf);
	ELSE
	Setpoint_SteamFan_IN:= Setpoint_SteamFan_Visu;
	END_IF

	SteamFAN_Switch_ON:=SteamFAN_Switch_ON_manu;
	SteamFan_ON:=SteamFan_ON_manu;





	Heat_matt1:=(Heat_matt1_manu ) AND Heat_Matt11_OK_for_heat ;
	Heat_matt2:=(Heat_matt2_manu  ) AND Heat_Matt2_OK_for_heat ;
	Heat_matt3:=(Heat_matt3_manu  ) AND Heat_Matt3_OK_for_heat ;
	Heat_matt4:=(Heat_matt4_manu  ) AND Heat_Matt4_OK_for_heat ;
	Heat_matt5:=(Heat_matt5_manu ) AND Heat_Matt5_OK_for_heat ;
	Heat_matt6:=(Heat_matt6_manu ) AND Heat_Matt6_OK_for_heat ;
	Heat_matt7:=(Heat_matt7_manu ) AND Heat_Matt7_OK_for_heat ;
	Heat_matt8:=(Heat_matt8_manu ) AND Heat_Matt8_OK_for_heat ;
	Heat_matt9:=(Heat_matt9_manu ) AND Heat_Matt9_OK_for_heat ;
	Heat_matt10:=(Heat_matt10_manu ) AND Heat_Matt10_OK_for_heat ;



	HEAT_Reg_1_OUT:=HEAT_Reg_1_manu;
	HEAT_Reg_2_OUT:=HEAT_Reg_2_manu;
	HEAT_Reg_3_OUT:=HEAT_Reg_3_manu;
	HEAT_Reg_4_OUT:=HEAT_Reg_4_manu;
	HEAT_Reg_5_OUT:=HEAT_Reg_5_manu;
	HEAT_Reg_6_OUT:=HEAT_Reg_6_manu;
	HEAT_Reg_7_OUT:=HEAT_Reg_7_manu;
	HEAT_Reg_8_OUT:=HEAT_Reg_8_manu;






	HEAT_Reg_Mainswitch_out:=HEAT_Reg_Mainswitch_manu;


	(* Wichtig!!! Hier werden beim einschalten in Manubetrieb für einen Puls die Ventile in die Startposition gesteuert*)


		Start_Puls_Valves:=TRUE;
		R_TRIG13(CLK:=Start_Puls_Valves , Q=>Start_Puls_Valves_out );
		
		IF Start_Puls_Valves_out  THEN

		V_Dampf_nach_Komp_manu:=FALSE; (*VE_K2.71*)
		V_Nach_WT_manu:=FALSE;  (*VE_K2.73*)
		V_Entlueftung_1_manu:=FALSE;  (*VExx*)
		V_Entlueftung_2_manu:=FALSE;  (*VExx*)
		V_Global_Res_3_manu:=FALSE;  (*VExx*)
		V_Global_Res_4_manu:=FALSE;  (*VExx*)
		V_Global_Res_5_manu:=FALSE;  (*VExx*)

		END_IF;



	(*Wichtig!! Zurzeit ist ganz unten die verknüpfen von den Ventil-Ausgängen. Dort werden die Sequence und Manu Befehle als SR-Glied zusammengefasst*)


	




(*_________________________________________________________________________________________CONTROL___AUTO____________________________________________*)
 ELSE IF Control_Auto_active THEN


Compressor_cooling:=Compressor_cooling_auto;

(*MAcht meiner Meinung nach zurzeit keinen Sinn die Reglersollwerte im OP Auto glechzusetzten wie im MANU OP, einfach mit aktiviertem Controller-Switch*)
(*
Setpoint_Compressor_IN:=REAL_TO_INT(fStellwert_comp); (*1.  ev noch die Ausgangsvariablen auf REAL setzten bezgtl  Genauigkeit			2. Setpoint_Compressor_Auto;___zurzeit nicht benötigt*)
Setpoint_Primaer_Comp_IN:=REAL_TO_INT(fStellwert_Primaer_Comp);
*)


Setpoint_Fan_IN:=Setpoint_Fan_Auto;
Setpoint_SteamFan_IN:=Setpoint_SteamFan_Auto;


Setpoint_M_Belts_IN:=Setpoint_M_Belts_Auto;
Setpoint_M_Belt_Feeder_IN:=Setpoint_M_Belt_Feeder_Auto;

Steamgenerator:=Steamgenerator_auto;




HEAT_Reg_Mainswitch_out:=HEAT_Reg_Mainswitch_auto;









(*
V_Dampf_nach_Komp (*VE_K2.71*)
V_Nach_WT (*VE_K2.73*)
V_Entlueftung_1 (*VE_Kxxx*)
V_Entlueftung_2 (*VE_Kxxx*)
V_Global_Res_3 (*VE_Kxxx*)
V_Global_Res_4 (*VE_Kxxx*)
V_Global_Res_5 (*VE_Kxxx*)

*)


V_Dampf_nach_Komp:=V_Dampf_nach_Komp_auto;
V_Nach_WT:=V_Nach_WT_auto;
V_Entlueftung_1:=V_Entlueftung_1_auto;
V_Entlueftung_2:=V_Entlueftung_2_auto;
V_Global_Res_3:=V_Global_Res_3_auto;
V_Global_Res_4:=V_Global_Res_4_auto;
V_Global_Res_5:=V_Global_Res_5_auto;







ELSE


	Start_Puls_Valves:=FALSE;
	Heat_matt1_manu:=FALSE;
	Heat_matt2_manu:=FALSE;
	Heat_matt3_manu:=FALSE;
	Heat_matt4_manu:=FALSE;
	Heat_matt5_manu:=FALSE;
	Heat_matt6_manu:=FALSE;
	Heat_matt7_manu:=FALSE;
	Heat_matt8_manu:=FALSE;
	Heat_matt9_manu:=FALSE;
	Heat_matt10_manu:=FALSE;
	Heat_matt1_auto:=FALSE;
	Heat_matt2_auto:=FALSE;
	Heat_matt3_auto:=FALSE;
	Heat_matt4_auto:=FALSE;
	Heat_matt5_auto:=FALSE;
	Heat_matt6_auto:=FALSE;
	Heat_matt7_auto:=FALSE;
	Heat_matt8_auto:=FALSE;
	Heat_matt9_auto:=FALSE;
	Heat_matt10_auto:=FALSE;
	
	Heat_matt_Group1_1_4_auto:=FALSE;
	Heat_matt_Group2_5_8_auto:=FALSE;
	Heat_matt_Group3_9_10_auto:=FALSE;
	
	Heat_matt1:=FALSE;
	Heat_matt2:=FALSE;
	Heat_matt3:=FALSE;
	Heat_matt4:=FALSE;
	Heat_matt5:=FALSE;
	Heat_matt6:=FALSE;
	Heat_matt7:=FALSE;
	Heat_matt8:=FALSE;
	Heat_matt9:=FALSE;
	Heat_matt10:=FALSE;
	
	Heat_matt_Group1_1_4:=FALSE;
	Heat_matt_Group2_5_8:=FALSE;
	Heat_matt_Group3_9_10:=FALSE;




	HEAT_Reg_1_OUT:=FALSE;
	HEAT_Reg_2_OUT:=FALSE;
	HEAT_Reg_3_OUT:=FALSE;
	HEAT_Reg_4_OUT:=FALSE;
	HEAT_Reg_5_OUT:=FALSE;
	HEAT_Reg_6_OUT:=FALSE;
	HEAT_Reg_7_OUT:=FALSE;
	HEAT_Reg_8_OUT:=FALSE;




	HEAT_Reg_Mainswitch_out:=FALSE;

	HEAT_Reg_1_auto:=FALSE;
	HEAT_Reg_2_auto:=FALSE;
	HEAT_Reg_3_auto:=FALSE;
	HEAT_Reg_4_auto:=FALSE;
	HEAT_Reg_5_auto:=FALSE;
	HEAT_Reg_6_auto:=FALSE;
	HEAT_Reg_7_auto:=FALSE;
	HEAT_Reg_8_auto:=FALSE;



	HEAT_Reg_Mainswitch_auto:=FALSE;

	HEAT_Reg_1_Manu:=FALSE;
	HEAT_Reg_2_Manu:=FALSE;
	HEAT_Reg_3_Manu:=FALSE;
	HEAT_Reg_4_Manu:=FALSE;
	HEAT_Reg_5_Manu:=FALSE;
	HEAT_Reg_6_Manu:=FALSE;
	HEAT_Reg_7_Manu:=FALSE;
	HEAT_Reg_8_Manu:=FALSE;


	HEAT_Reg_Mainswitch_Manu:=FALSE;




	bManuHeat_REG1_CTRL:=FALSE;
	bManuHeat_REG2_CTRL:=FALSE;
	bManuHeat_REG3_CTRL :=FALSE;
	bManuHeat_REG4_CTRL :=FALSE;
	bManuHeat_REG5_CTRL:=FALSE;
	bManuHeat_REG6_CTRL:=FALSE;
	bManuHeat_REG7_CTRL :=FALSE;
	bManuHeat_REG8_CTRL :=FALSE;


	(*bManu_Heat_EinschraubHZK1_CTRL:=FALSE;
	bManu_Heat_EinschraubHZK2_CTRL:=FALSE;
	bManu_Heat_EinschraubHZK3_CTRL:=FALSE;
	bManu_Heat_REG_Comp:=FALSE;*)








	V_Dampf_nach_Komp:=FALSE;
	V_Nach_WT:=FALSE;
	V_Entlueftung_1:=FALSE;
	V_Entlueftung_2:=FALSE;
	V_Global_Res_3:=FALSE;
	V_Global_Res_4:=FALSE;
	V_Global_Res_5:=FALSE;



	V_Dampf_nach_Komp_auto:=FALSE;
	V_Nach_WT_auto:=FALSE;
	V_Entlueftung_1_auto:=FALSE;
	V_Entlueftung_2_auto:=FALSE;
	V_Global_Res_3_auto:=FALSE;
	V_Global_Res_4_auto:=FALSE;
	V_Global_Res_5_auto:=FALSE;


	V_Dampf_nach_Komp_manu:=FALSE;
	V_Nach_WT_manu:=FALSE;
	V_Entlueftung_1_manu:=FALSE;
	V_Entlueftung_2_manu:=FALSE;
	V_Global_Res_3_manu:=FALSE;
	V_Global_Res_4_manu:=FALSE;
	V_Global_Res_5_manu:=FALSE;




	FAN_Switch_ON:=FALSE;
	FAN_ON:=FALSE;
	FAN_Switch_ON_Manu:=FALSE;
	FAN_ON_Manu:=FALSE;

	Compressor_Switch_ON:=FALSE;
	Compressor_ON:=FALSE;
	Compressor_Switch_ON_manu:=FALSE;
	Compressor_ON_manu:=FALSE;

	Compressor_cooling_manu :=FALSE;
	Compressor_cooling_auto :=FALSE;
	Compressor_cooling :=FALSE;

	SteamFAN_Switch_ON:=FALSE;
	SteamFAN_Switch_ON_Manu:=FALSE;
	SteamFan_ON:=FALSE;
	SteamFan_ON_manu:=FALSE;


	M_Belts_ON:=FALSE;
	M_Belts_Switch_ON:=FALSE;
	M_Belts_Switch_ON_Manu:=FALSE;
	M_Belts_ON_Manu:=FALSE;


	M_Belt_Feeder_ON:=FALSE;
	M_Belt_Feeder_Switch_ON:=FALSE;
	M_Belt_Feeder_Switch_ON_Manu:=FALSE;
	M_Belt_Feeder_ON_Manu:=FALSE;



END_IF
END_IF





(*____________________________________________________________________AUTOSTART___________________________________________________*)

(*



R_TRIG12(CLK:= OK_continue_Austostartup_VISU, Q=>OK_continue_Austostartup );


(*Zeiten für Startphase: T21-T26 zurzeit : T21 2Sek. T22 10s*)

IF Auto_Startup AND Cabinet_OK  AND Des_Main_Aktive = FALSE AND ADS_Main_Aktive =FALSE  THEN

Startup_Active:=TRUE;

CASE C_Startup OF

0:
	String_Startup:='';
	IN_T21:=FALSE;
	IN_T22:=FALSE;
	C_Startup:=1;

1:
	Compressor_Switch_ON_Manu:=TRUE;
	Set_Valve_Sequence_Default:=TRUE;
	LED_green_VISU:=FALSE;
	LED_yellow_VISU:=TRUE;
	LED_RED_VISU:=FALSE;
	LED_white_VISU:=FALSE;

	Valve_Water_Out_manu:=TRUE;	(*_____________Austauschen___________________*)
	Valve_Air_Release_manu:=TRUE;	(*_____________Austauschen___________________*)

	IN_T21:=TRUE;
	C_Startup:=2;
2:
	IF Compressor_OK AND OUT_T21 THEN
	Set_Valve_Sequence_Default:=FALSE;
	Valve_Vacuum_breaker1_manu:=TRUE;
	Valve_Vacuum_breaker2_manu:=TRUE;
	Valve_SG_manu:=TRUE;
	IN_T21:=FALSE;
	Setpoint_Compressor_Visu:=50;
	Compressor_ON_Manu:=TRUE;
	C_Startup:=3;
	ELSE
	C_Startup:=2;
	END_IF;

	3:C_Startup:=4;
	4:C_Startup:=5;
	5:C_Startup:=6;
	6:C_Startup:=7;

7:
	Valve_ST_back_manu:=TRUE;	(*_____________Austauschen___________________*)
	Valve_SG_manu:=FALSE;	(*_____________Austauschen___________________*)

	IN_T21:=TRUE;
	C_Startup:=8;

8:	C_Startup:=9;
9:	C_Startup:=10;

10:
	IF OUT_T21 THEN
	IN_T21:=FALSE;
	Valve_ST_back_manu:=FALSE;	(*_____________Austauschen___________________*)
	Switch_Heat_group1:=TRUE;
	Switch_Heat_group2 :=TRUE;
	Switch_Heat_group3 :=TRUE;
	Heat_matt_Group1_1_4_manu:=TRUE;
	Heat_matt_Group2_5_8_manu:=TRUE;
	Heat_matt_Group3_9_10_manu:=TRUE;

	C_Startup:=11;
	ELSE
	C_Startup:=10;
	END_IF;

11:	IN_T21:=TRUE;
	C_Startup:=12;

12:
	IF OUT_T21 THEN
	IN_T21:=FALSE;
	C_Startup:=13;

	String_Startup:='Please switch on control Panel Steam Generator';

	ELSE
	C_Startup:=12;
	END_IF;

13:
	IF OK_continue_Austostartup THEN

	String_Startup:='Waiting for Steam is hot';

	C_Startup:=14;
	ELSE
	C_Startup:=13;
	END_IF;

14:
	IF OK_continue_Austostartup THEN

	Set_Valve_Sequence_Default:=TRUE;

	String_Startup:='Preaparing for Steam Inlet compressor';

	C_Startup:=15;
	ELSE
	C_Startup:=14;
	END_IF;

15:
	IF OK_continue_Austostartup THEN
	Set_Valve_Sequence_Default:=FALSE;
	String_Startup:='Waiting for temp. Compressor';
	IN_T22:=FALSE;
	C_Startup:=16;
	ELSE
	C_Startup:=15;
	END_IF;

16:
	Check_compressor_Temp:=TRUE;
	IF Temp_compressor_Self > 60 OR Temp_compressor > 100 THEN
	IN_T22:=TRUE;
	C_Startup:=17;
	ELSE
	C_Startup:=16;
	END_IF;

17:
	IF Temp_compressor_Self > 60 OR Temp_compressor > 100 AND OUT_T22 THEN
	Valve_ST_back_manu:=FALSE;	(*_____________Austauschen___________________*)
	IN_T22:=FALSE;
	Setpoint_Compressor_Visu:=85;
	Check_compressor_Temp:=FALSE;
	String_Startup:='Steam Inlet in the next seconds!!!';
	C_Startup:=18;
	ELSE
	C_Startup:=17;
	END_IF;

18:	IN_T22:=TRUE;
	C_Startup:=19;

19:
	IF OUT_T22 THEN
	String_Startup:='Steam Inlet OK';
	IN_T21:=FALSE;
	IN_T22:=FALSE;
(*
	Valv_SG_Seqence:=TRUE;
	Valve_Air_IN_Seqence:=TRUE;
	Valve_ST_IN_Seqence:=TRUE;
	Valve_Comp_IN_Seqence:=TRUE;
	Valve_ST_back_Seqence:=FALSE;
	Valve_Water_Out_Seqence:=TRUE;*)

	(*_____________Austauschen___________________*)

	C_Startup:=20;
	ELSE
	C_Startup:=19;
	END_IF;

	20:C_Startup:=21;
	21:C_Startup:=22;
	22:C_Startup:=23;
	23:C_Startup:=24;
	24:C_Startup:=25;
	25:C_Startup:=26;
	26:C_Startup:=43;





43:	Startup_Finished:=TRUE;

END_CASE


ELSE

Startup_Finished:=FALSE;

(* Ausschaltimpuls*)
F_TRIG10(CLK:=Startup_Active);
IF F_TRIG10.Q THEN
LED_yellow_VISU:=FALSE;
LED_RED_VISU:=FALSE;
LED_white_VISU:=FALSE;
Valve_ST_back_manu:=FALSE;
END_IF;

Startup_Active:=FALSE;
C_Startup:=0;
Check_compressor_Temp:=FALSE;
END_IF;


*)

























(* ___Dieser Bereich wird zurzeit NICHT benötigt!!!








(*________________________________________________________________________Start Adsorbtion__________________________________________________________*)


IF ADS_active =FALSE  THEN
C_ADS:=0;
ADS_Main_Aktive:=FALSE;
END_IF





CASE C_ADS OF

0:	IN_T4:=FALSE;
	IN_T5:=FALSE;
	IN_T6:=FALSE;
	IN_T7:=FALSE;
	IN_T8:=FALSE;
	IN_T9:=FALSE;
	(*Desorbtion_complete:=FALSE;*)
	Weight_Sample1_OK:=FALSE;
	TIME_DONE_ADS:=FALSE;
	ADS_Main_Aktive:=FALSE;
	Setpoint_Fan_Auto:=0;
	Valvematrix:=0;
	C_ADS:=1;

1:
	(*Bedingungen zum Start: 1. OK von Not-Aus Relais 2. OK von Gewichtsangbaen...... *)

	IF   Cabinet_OK  AND Start_ADS AND DES_active=FALSE  THEN
	ADS_Main_Aktive:=TRUE;
	Compressor_Switch_ON:=FALSE;
	Compressor_ON:=FALSE;
	FAN_Switch_ON:=TRUE;
	FAN_ON:=TRUE;
	IN_T6:=TRUE;


		IF OUT_T6 THEN
		IN_T6:=FALSE;
		Setpoint_Fan_Auto:=20; (* (%) Wert Ändern*)
		C_ADS:=2;
		END_IF

	ELSE
	C_ADS:=1;
	END_IF

2:
	(*Zeit starten ADS*)
	C_ADS:=3;
	IN_T4:=TRUE;

(* Entweder ist die die Bedingung zum beenden der Adsorption die Zeit oder das Gewicht*)

3:
	IF OUT_T4  THEN

		IN_T4:=FALSE;
		IN_T6:=TRUE;
		TIME_DONE_ADS:=TRUE;
		Setpoint_Fan_Auto:=0;
		C_ADS:=4;


	ELSE IF  	Weight_OK (* WERT GEàNDERT WREDEN!!!!!!!!!!!!!!!!!!!!!!!!!!!!!!!!!!!!!!!!!!!!!!!!!*) THEN

		(*Weight_Sample1_OK:=TRUE;*)
		IN_T4:=FALSE;
		IN_T6:=TRUE;
		C_ADS:=4;
		Setpoint_Fan_Auto:=0;
		ELSE
		C_ADS:=3;

	END_IF
	END_IF


4:	IF OUT_T6 THEN
	IN_T6:=FALSE;
	ADS_Main_Aktive:=FALSE;
	TIME_DONE_ADS:=FALSE;
	C_ADS:=5;
	ELSE
	C_ADS:=4;
	END_IF





6:	C_ADS:=7;
7:	C_ADS:=100;
100:	C_ADS:=0;


END_CASE




(* Zusätzliches ADSORBTION
*)


(* Wenn Wage 2 nach WT anfängt weniger aufzunhemen wie Wage 1 dann ist die Schüttung langsam voll*)

Weight_DIFF:=Weight_Sample1-Weight_Sample2;





*)



























(*___________________________________________________Allg. Hysteresen_________________________________________________________________*)







(*Hyterese Temp. Kompressor*)
IF Temp_compressor_Self > Limit_Temp_Compressor THEN IN_T100:=TRUE; ELSE IF Temp_compressor_Self < Limit_Temp_Compressor THEN IN_T100:=FALSE; END_IF END_IF
IF OUT_T100 THEN Temp_compressor_OK:=TRUE; ELSE Temp_compressor_OK:=FALSE; END_IF

(*
(*Hyterese Temp. Verdampfegehäuse  Es wird der Durchschnitt aller 4 Temp. sensoren abgefragt*)
IF Temp_Cabinet_averange > Limit_Temp_Cabinet  THEN IN_T102:=TRUE; ELSE IF Temp_Cabinet_averange < Limit_Temp_Cabinet THEN IN_T102:=FALSE; END_IF END_IF
IF OUT_T102 THEN Temp_Cabinet_OK:=TRUE; ELSE Temp_Cabinet_OK:=FALSE; END_IF

(*Hyterese Gehäuse abkühlern*)
IF Temp_Cabinet_averange < Limit_Temp_cooling_Cabinet  THEN IN_T103:=TRUE; ELSE IF Temp_Cabinet_averange   > Limit_Temp_cooling_Cabinet  THEN IN_T103:=FALSE; END_IF END_IF
IF OUT_T103 THEN Cooling_OK:=TRUE; ELSE Cooling_OK:=FALSE; END_IF

*)


(*Heizmatten 1-10*)



Hyst1(Hyst_Value:=Temp_Heatmatt1 , Hyst_Low_Limit:=Hyst_low_LIM_Heatmatt , Hyst_Hight_Limit:=Hyst_high_LIM_Heatmatt, Hyst_OUT=> Heat_Matt11_OK_for_heat );
Hyst2(Hyst_Value:=Temp_Heatmatt2 , Hyst_Low_Limit:=Hyst_low_LIM_Heatmatt , Hyst_Hight_Limit:=Hyst_high_LIM_Heatmatt , Hyst_OUT=> Heat_Matt2_OK_for_heat );
Hyst3(Hyst_Value:=Temp_Heatmatt3 , Hyst_Low_Limit:=Hyst_low_LIM_Heatmatt , Hyst_Hight_Limit:=Hyst_high_LIM_Heatmatt , Hyst_OUT=> Heat_Matt3_OK_for_heat );
Hyst4(Hyst_Value:=Temp_Heatmatt4 , Hyst_Low_Limit:=Hyst_low_LIM_Heatmatt , Hyst_Hight_Limit:=Hyst_high_LIM_Heatmatt , Hyst_OUT=> Heat_Matt4_OK_for_heat );
Hyst5(Hyst_Value:=Temp_Heatmatt5 , Hyst_Low_Limit:=Hyst_low_LIM_Heatmatt , Hyst_Hight_Limit:=Hyst_high_LIM_Heatmatt , Hyst_OUT=> Heat_Matt5_OK_for_heat );
Hyst6(Hyst_Value:=Temp_Heatmatt6 , Hyst_Low_Limit:=Hyst_low_LIM_Heatmatt , Hyst_Hight_Limit:=Hyst_high_LIM_Heatmatt , Hyst_OUT=> Heat_Matt6_OK_for_heat );
Hyst7(Hyst_Value:=Temp_Heatmatt7 , Hyst_Low_Limit:=Hyst_low_LIM_Heatmatt , Hyst_Hight_Limit:=Hyst_high_LIM_Heatmatt , Hyst_OUT=> Heat_Matt7_OK_for_heat );
Hyst8(Hyst_Value:=Temp_Heatmatt8 , Hyst_Low_Limit:=Hyst_low_LIM_Heatmatt , Hyst_Hight_Limit:=Hyst_high_LIM_Heatmatt , Hyst_OUT=> Heat_Matt8_OK_for_heat );
Hyst9(Hyst_Value:=Temp_Heatmatt9 , Hyst_Low_Limit:=Hyst_low_LIM_Heatmatt , Hyst_Hight_Limit:=Hyst_high_LIM_Heatmatt , Hyst_OUT=> Heat_Matt9_OK_for_heat );
Hyst10(Hyst_Value:=Temp_Heatmatt10 , Hyst_Low_Limit:=Hyst_low_LIM_Heatmatt , Hyst_Hight_Limit:=Hyst_high_LIM_Heatmatt , Hyst_OUT=> Heat_Matt10_OK_for_heat );



(*IF Temp_Heatmatt1> 120 THEN Heat_matt1:=FALSE; END_IF
IF Temp_Heatmatt2> 120 THEN Heat_matt2:=FALSE; END_IF
IF Temp_Heatmatt3> 120 THEN Heat_matt3:=FALSE; END_IF
IF Temp_Heatmatt4> 120 THEN Heat_matt4:=FALSE; END_IF
IF Temp_Heatmatt5> 120 THEN Heat_matt5:=FALSE; END_IF
IF Temp_Heatmatt6> 120 THEN Heat_matt6:=FALSE; END_IF
IF Temp_Heatmatt7> 120 THEN Heat_matt7:=FALSE; END_IF
IF Temp_Heatmatt8> 120 THEN Heat_matt8:=FALSE; END_IF
IF Temp_Heatmatt9> 120 THEN Heat_matt9:=FALSE; END_IF
IF Temp_Heatmatt10> 120 THEN Heat_matt10:=FALSE; END_IF

*)



END_IF













(*Zusätzliches*)



(*Ventilmatrix*)

(*
IF Valvematrix.0 =TRUE THEN Valve_YB1:=TRUE; ELSE Valve_YB1:=FALSE;END_IF;
IF Valvematrix.1 =TRUE THEN Valve_YB2:=TRUE; ELSE Valve_YB2:=FALSE; END_IF;
IF Valvematrix.2 =TRUE THEN Valve_YB3:=TRUE; ELSE Valve_YB3:=FALSE; END_IF;
IF Valvematrix.3 =TRUE THEN Valve_YB4:=TRUE; ELSE Valve_YB4:=FALSE; END_IF;
IF Valvematrix.4 =TRUE THEN Valve_YB6:=TRUE; ELSE Valve_YB6:=FALSE; END_IF;
IF Valvematrix.5 =TRUE THEN Valve_YB7:=TRUE; ELSE Valve_YB7:=FALSE; END_IF;
IF Valvematrix.6 =TRUE THEN Valve_YB8:=TRUE; ELSE Valve_YB8:=FALSE; END_IF;
Valve_YB9:=Valvematrix2.0;
Valve_YB10:=Valvematrix2.1;
*)



IF All_Heater_on_auto THEN
Heat_matt1_auto:=TRUE;
Heat_matt2_auto:=TRUE;
Heat_matt3_auto:=TRUE;
Heat_matt4_auto:=TRUE;
Heat_matt5_auto:=TRUE;
Heat_matt6_auto:=TRUE;
Heat_matt7_auto:=TRUE;
Heat_matt8_auto:=TRUE;
Heat_matt9_auto:=TRUE;
Heat_matt10_auto:=TRUE;
END_IF;









(*

Info: Zurzeit brauchts diese Modbus-Variablenzuweisung noch nicht, es wird versucht diesmal auf TC3 umzustellen inkl. Visu

WIchtig!!! Die Bez. IN OUT ist aus versehen verkehrt!!!!*)





(*


(*Modbusvariablenzuweiseung*)



 (*SPS seitig Eingänge*)

(*Binär:*)

(*Main_ON:=mb_Output_Coils[0];*)

(*Analog:*)


	Register_IN1:=mb_Output_Registers[0];
	Register_IN2:=mb_Output_Registers[1];
	Register_IN3:=mb_Output_Registers[2];
	Register_IN4:=mb_Output_Registers[3];
	Register_IN5:=mb_Output_Registers[4];
	Register_IN6:=mb_Output_Registers[5];
	Register_IN7:=mb_Output_Registers[6];
	Register_IN8:=mb_Output_Registers[7];
	Register_IN9:=mb_Output_Registers[8];
	Register_IN10:=mb_Output_Registers[9];


 (*SPS seitig Ausgänge*)

(*Binär:*)

mb_Input_Coils[0]:=V_Dampf_nach_Komp;
mb_Input_Coils[1]:=V_Nach_WT;
mb_Input_Coils[2]:=V_Entlueftung_1;
mb_Input_Coils[3]:=V_Entlueftung_2;
mb_Input_Coils[4]:=V_Global_Res_3;
mb_Input_Coils[5]:=V_Global_Res_4;
mb_Input_Coils[6]:=V_Global_Res_5;
mb_Input_Coils[7]:=V_Wasserauslass;
mb_Input_Coils[8]:=V_Dichtringe_Einlass;
mb_Input_Coils[9]:=V_Dichtringe_Auslass;
mb_Input_Coils[10]:=Compressor_PT100_Error;






(*Analog:*)

mb_Input_Registers[0]:=0;
mb_Input_Registers[1]:=0;
mb_Input_Registers[2]:=0;
mb_Input_Registers[3]:=0;
mb_Input_Registers[4]:=0;
mb_Input_Registers[5]:=0;
mb_Input_Registers[6]:=0;
mb_Input_Registers[7]:=0;
mb_Input_Registers[8]:=0;
mb_Input_Registers[9]:=0;
mb_Input_Registers[10]:=REAL_TO_INT(T_Vor_DecicWheel*100);		(*Zur Info::: Zurzeit sollen NUR die Temps mit Faktor 100 transferiert werden, da sonst bei den Drücken mit Milibarausdruck ein Overflow des Wertes wäre*)
mb_Input_Registers[11]:=REAL_TO_INT(T_Nach_DecicWheel*100);
mb_Input_Registers[12]:=REAL_TO_INT(T_Des_nach_V_Umdampf*100);
mb_Input_Registers[13]:=REAL_TO_INT(T_Des_nach_WT*100);
mb_Input_Registers[14]:=REAL_TO_INT(T_Des_vor_DecicWheel*100);
mb_Input_Registers[15]:=REAL_TO_INT(T_comp_gehause*100);
mb_Input_Registers[16]:=REAL_TO_INT(T_Dampfleitung_comp*100);
mb_Input_Registers[17]:=REAL_TO_INT(T_Vor_KlauenkolbenKomp*100);(*T3.31*)
mb_Input_Registers[18]:=REAL_TO_INT(T_Windfenster_IMDampf_oben*100);
mb_Input_Registers[19]:=REAL_TO_INT(T_Windfenster_IMDampf_unten*100);
mb_Input_Registers[20]:=REAL_TO_INT(9999);
mb_Input_Registers[21]:=REAL_TO_INT(T_Wasserwanne*100);
mb_Input_Registers[22]:=REAL_TO_INT(Temp_Heatmatt1*100);
mb_Input_Registers[23]:=REAL_TO_INT(Temp_Heatmatt2*100);
mb_Input_Registers[24]:=REAL_TO_INT(Temp_Heatmatt3*100);
mb_Input_Registers[25]:=REAL_TO_INT(Temp_Heatmatt4*100);
mb_Input_Registers[26]:=REAL_TO_INT(Temp_Heatmatt5*100);
mb_Input_Registers[27]:=REAL_TO_INT(Temp_Heatmatt6*100);
mb_Input_Registers[28]:=REAL_TO_INT(Temp_Heatmatt7*100);
mb_Input_Registers[29]:=REAL_TO_INT(Temp_Heatmatt8*100);
mb_Input_Registers[30]:=REAL_TO_INT(Temp_Heatmatt9*100);
mb_Input_Registers[31]:=REAL_TO_INT(Temp_Heatmatt10*100);
mb_Input_Registers[32]:=REAL_TO_INT(T_Ambiente*100);
mb_Input_Registers[33]:=REAL_TO_INT(T_Einlass_Kompressor*100); 	(*SET 3.33*)
mb_Input_Registers[34]:=REAL_TO_INT(T_Heizband_Filter2*100);
mb_Input_Registers[35]:=REAL_TO_INT(T_Heizband_Filter3*100);
mb_Input_Registers[36]:=REAL_TO_INT(T_Monitor_Heatreg1*100);
mb_Input_Registers[37]:=REAL_TO_INT(T_Monitor_Heatreg2*100);
mb_Input_Registers[38]:=0;
mb_Input_Registers[39]:=0;
mb_Input_Registers[40]:=REAL_TO_INT(RH_Vor_DecicWheel*100);
mb_Input_Registers[41]:=REAL_TO_INT(RH_Nach_DecicWheel*100);
mb_Input_Registers[42]:=REAL_TO_INT(RH_Des_nach_V_Umdampf*100);
mb_Input_Registers[43]:=REAL_TO_INT(RH_Des_nach_WT*100);
mb_Input_Registers[44]:=0;
mb_Input_Registers[45]:=0;
mb_Input_Registers[46]:=0;
mb_Input_Registers[47]:=0;
mb_Input_Registers[48]:=0;
mb_Input_Registers[49]:=0;
mb_Input_Registers[50]:=REAL_TO_INT(P_Des_nach_V_Umdampf);
mb_Input_Registers[51]:=REAL_TO_INT(P_Des_nach_WT);
mb_Input_Registers[52]:=REAL_TO_INT(P_Dampfleitung_comp);
mb_Input_Registers[53]:=REAL_TO_INT(P_Vor_KlauenkolbenKomp);
mb_Input_Registers[54]:=REAL_TO_INT(P_Windfenster_1);
mb_Input_Registers[55]:=REAL_TO_INT(P_Windfenster_2);
mb_Input_Registers[56]:=REAL_TO_INT(P_Drucklufttank);
mb_Input_Registers[57]:=REAL_TO_INT(P_Sperrgasdichtung);
mb_Input_Registers[58]:=REAL_TO_INT(P_Amb);
mb_Input_Registers[59]:=REAL_TO_INT(P_Zwischenstufe_Kompressoren);
mb_Input_Registers[60]:=REAL_TO_INT(Ps_311);
mb_Input_Registers[61]:=REAL_TO_INT(Ps_26);
mb_Input_Registers[62]:=REAL_TO_INT(Ps_28);
mb_Input_Registers[63]:=0;
mb_Input_Registers[64]:=0;
mb_Input_Registers[65]:=0;
mb_Input_Registers[66]:=0;
mb_Input_Registers[67]:=0;
mb_Input_Registers[68]:=0;
mb_Input_Registers[69]:=0;
mb_Input_Registers[70]:=REAL_TO_INT(RelP_TM*100);
mb_Input_Registers[71]:=REAL_TO_INT(RelP_WT*100);
mb_Input_Registers[72]:=REAL_TO_INT(RelP_OUT*100);
mb_Input_Registers[73]:=0;
mb_Input_Registers[74]:=0;
mb_Input_Registers[75]:=0;
mb_Input_Registers[76]:=0;
mb_Input_Registers[77]:=0;
mb_Input_Registers[78]:=0;
mb_Input_Registers[79]:=0;
mb_Input_Registers[80]:=REAL_TO_INT(Current_OUT_SteamVenti_L1*100);
mb_Input_Registers[81]:=REAL_TO_INT(Current_OUT_SteamVenti_L2*100);
mb_Input_Registers[82]:=REAL_TO_INT(Current_OUT_SteamVenti_L3*100);
mb_Input_Registers[83]:=REAL_TO_INT(Current_OUT_HEAT_Reg_1*100);
mb_Input_Registers[84]:=REAL_TO_INT(Current_OUT_HEAT_Reg_2*100);
mb_Input_Registers[85]:=REAL_TO_INT(Current_OUT_HEAT_Reg_3*100);
mb_Input_Registers[86]:=REAL_TO_INT(Current_OUT_HEAT_Reg_4*100);
mb_Input_Registers[87]:=REAL_TO_INT(Current_OUT_Compressor_L1 *100);
mb_Input_Registers[88]:=REAL_TO_INT(Current_OUT_Compressor_L2 *100);
mb_Input_Registers[89]:=REAL_TO_INT(Current_OUT_Compressor_L3 *100);
mb_Input_Registers[90]:=REAL_TO_INT(Current_OUT_AdsorbtionsVenti_L1 *100);
mb_Input_Registers[91]:=REAL_TO_INT(Current_OUT_AdsorbtionsVenti_L2 *100);
mb_Input_Registers[92]:=REAL_TO_INT(Current_OUT_AdsorbtionsVenti_L3 *100);
mb_Input_Registers[93]:=REAL_TO_INT(Current_OUT_Fan_L1*100);
mb_Input_Registers[94]:=REAL_TO_INT(Current_OUT_Fan_L2 *100);
mb_Input_Registers[95]:=REAL_TO_INT(Current_OUT_Fan_L3*100);
mb_Input_Registers[96]:=REAL_TO_INT(Current_OUT_Complete_L1 *100);
mb_Input_Registers[97]:=REAL_TO_INT(Current_OUT_Complete_L2 *100);
mb_Input_Registers[98]:=REAL_TO_INT(Current_OUT_Complete_L3 *100);
mb_Input_Registers[99]:=0;
mb_Input_Registers[100]:=0;
mb_Input_Registers[101]:=0;
mb_Input_Registers[102]:=0;
mb_Input_Registers[103]:=0;
mb_Input_Registers[104]:=0;
mb_Input_Registers[105]:=0;
mb_Input_Registers[106]:=0;
mb_Input_Registers[107]:=0;
mb_Input_Registers[108]:=0;
mb_Input_Registers[109]:=0;
mb_Input_Registers[110]:=0;
mb_Input_Registers[111]:=0;
mb_Input_Registers[112]:=0;
mb_Input_Registers[113]:=0;
mb_Input_Registers[114]:=0;
mb_Input_Registers[115]:=0;
mb_Input_Registers[116]:=0;
mb_Input_Registers[117]:=0;
mb_Input_Registers[118]:=0;
mb_Input_Registers[119]:=0;
mb_Input_Registers[120]:=REAL_TO_INT(Compressor_Actual_Turn);
mb_Input_Registers[121]:=REAL_TO_INT(SteamFan_Actual_Turn);	(*Muss dann wieder getauscgt werden, wenn ATV32 wieder für den Umdampfventi kommt*)
mb_Input_Registers[122]:=REAL_TO_INT(FAN_Actual_Turn);

*)




























(*________________MODBUS Server_______________________*)

IF NOT bWriteRegs THEN


	bWriteRegs :=TRUE;

	fbWriteRegs.sIPAddr :=ipAddr;
	fbWriteRegs.nQuantity := 7;
	nUnitID:=nUnitID;
	nTCPPort:=503;
	fbWriteRegs.nMBAddr := 16#200;	(*Offsetadresse*)
	fbWriteRegs.cbLength := SIZEOF(nValue);
	fbWriteRegs.pSrcAddr := ADR(nValue);
	fbWriteRegs.tTimeout := T#5s;
	fbWriteRegs(bExecute:=TRUE);
	bError:=fbWriteRegs.bError;
	nErrID:=fbWriteRegs.nErrID;
ELSE
	IF  NOT fbWriteRegs.bBUSY THEN
		bWriteRegs :=FALSE;
	END_IF
	fbWriteRegs(bExecute:=FALSE);
END_IF

nValue[0]:=10000; 	(*Periode of PWM Pokeys*)
nValue[6]:=PWM_duty_cycle*100; 	(*Duty Cycle*)




(*

PWM registers accept raw PWM duty cycle timer value - 
the resulting duty cycle is therefore the value of the duty register divided by the PWM period value. 
Two consecutive 16-bit registers make up the 32-bit PWM duty cycle register, so you must write both.*)

(*
die 200,203 sind bytes

200,201 PWM PERIOD (MSB first)
202,203 PWM duty1 (MSB first) – pin 22 ...
212,213 PWM duty6 (MSB first) – pin 17
*)






(*

WICHTIG!!!!!!!!!!!!! OFFSET vomModbus Client (MAster) ist immer 32768

Hier die EInstellungen im IAS:

Read Input Registers (FC04)	32768
Read Input Registers (FC04)	32769
Read Input Registers (FC04)	32770
Read Input Registers (FC04)	32771
Read Input Registers (FC04)	32772
Preset Single Register (FC06)	32768
Preset Single Register (FC06)	32769
Force Single Coil (FC05)	32768
Force Single Coil (FC05)	32769
Force Single Coil (FC05)	32770
Read Input Status (FC02)	0


*)


IF Start_Auto_Export_OUT THEN
Start_Auto_Export_INT:=1;
ELSE
Start_Auto_Export_INT:=0;
END_IF;





(*____________________________________________________________________________________________SIcherheiten________________________________________________________*)






(*SIcherheit, dass   bei hohem Dampfdruck öffnet*)
(*
IF P_OUT_Steamgenerator > P_Steamgenerator_to_big  THEN
Valve_SG_Preasure_release_manu;
END_IF
*)





IF Compressor_Switch_ON_Manu = FALSE OR Compressor_ON_Manu = FALSE THEN
Setpoint_Compressor_Visu:=0;
END_IF;



IF M_Belts_Switch_ON_Manu = FALSE OR M_Belts_ON_Manu = FALSE THEN
Setpoint_M_Belts_Visu:=0;
END_IF;


IF M_Belt_Feeder_Switch_ON_Manu = FALSE OR M_Belt_Feeder_ON_Manu = FALSE THEN
Setpoint_M_Belt_Feeder_Visu:=0;
END_IF;






(*IF SteamFAN_Switch_ON_manu = FALSE OR SteamFAN_Switch_ON_Manu = FALSE THEN
Setpoint_SteamFAN_Visu:=0;
END_IF;*)



IF FAN_Switch_ON_Manu = FALSE OR FAN_ON_Manu = FALSE  OR SteamFan_PTC_Error THEN
Setpoint_FAN_Visu:=0;
END_IF;

















(* Zeiten ALLGEMEIN *)


TON1(IN:=IN_T1 , PT:=t#1s, Q=>OUT_T1 , ET=> ); (*ZEIT Hauptschütz einschalten*)

TON2(IN:=IN_T2 , PT:=t#4s, Q=>OUT_T2 , ET=> ); (*ZEIT Überwachung Hauptschütz einschalten*)

TON3(IN:=IN_T3 , PT:=t#200s, Q=>OUT_T3 , ET=>ET_T3 );	(*Zeit für Stellanzeige Prop-  Kugelhhan orange*)



(*TON4-20 Frei! *)





(*Aufstartphase*)



TON21(IN:=IN_T21 , PT:=t#2s, Q=>OUT_T21 , ET=> );	(*Zeit für *)

TON22(IN:=IN_T22 , PT:=t#2s, Q=>OUT_T22 , ET=> );	(*Zeit für *)

TON23(IN:=IN_T23 , PT:=t#2s, Q=>OUT_T23 , ET=> );	(*Zeit für *)

TON24(IN:=IN_T24 , PT:=t#2s, Q=>OUT_T24 , ET=> );	(*Zeit für *)

TON25(IN:=IN_T25 , PT:=t#2s, Q=>OUT_T25 , ET=> );	(*Zeit für *)

TON26(IN:=IN_T26 , PT:=t#2s, Q=>OUT_T26 , ET=> );	(*Zeit für *)



























(* Hysterese DES*)


TON100(IN:=IN_T100 , PT:=T#10s, Q=>OUT_T100 , ET=> );	(*Hyst. aufheizen Kompressor*)
TON101(IN:=IN_T101 , PT:=T#10s, Q=>OUT_T101 , ET=> );	(*Hyst. erhitzen Wärmetauscher *)
TON102(IN:=IN_T102 , PT:=T#10s, Q=>OUT_T102, ET=> );	(*Hyst. Dampfgehäuse*)
TON103(IN:=IN_T103 , PT:=T#10s, Q=>OUT_T103 , ET=> );	(*Hyst.  Gehäuse abkühlen*)
TON104(IN:=IN_T104 , PT:=T#10s, Q=>OUT_T104 , ET=> );	(*Hyst.  RES*)
TON105(IN:=IN_T105 , PT:=T#10s, Q=>OUT_T105 , ET=> );	(*Hyst.  RES*)
TON106(IN:=IN_T106 , PT:=T#10s, Q=>OUT_T106 , ET=> );	(*Hyst.  RES*)
TON107(IN:=IN_T107 , PT:=T#10s, Q=>OUT_T107 , ET=> );	(*Hyst.  RES*)
TON108(IN:=IN_T108 , PT:=T#10s, Q=>OUT_T108 , ET=> );	(*Hyst.  RES*)
























(*

CTU1(
	CU:= C_up1,
	RESET:= Res_C1,
	PV:=,
	Q=> ,
	CV=> C_val1 );



CTU2(
	CU:= C_up2,
	RESET:= Res_C2,
	PV:= C_val2,
	Q=> ,
	CV=> );



CTU3(
	CU:= C_up3,
	RESET:= Res_C3,
	PV:= C_val3,
	Q=> ,
	CV=> );

*)

(*Reserve*)

CTU4(
	CU:= C_up4,
	RESET:= Res_C4,
	PV:= C_val4,
	Q=> ,
	CV=> );



F_TRIG1(CLK:=Control_Manu_active , Q=>OUT_FTRIG1 );




(*Bei dieser einfachen Variante eines PWM wird nach einem Taktmerkersignal (Pulsgen) eine Pulszeit (TP) dazugeschalten*)

IF Pulse2_set_manu THEN

Puls_GEN_Watervalve(bStart:=Enable_Pulsgen2 , tTakt:=REAL_TO_TIME(T_HI_Pulsegen2*1000 ), bBlink=>OUT_Pulsgen  );
Ton_Pulsgen(IN:=OUT_Pulsgen , PT:= REAL_TO_TIME(T_Pulstime_Pulsegen2*1000 ), Q=>Valve_YB7 , ET=> );

END_IF;





(*Umschaltmechanismen und Übergaben Ventile*)



IF V_Dampf_nach_Komp THEN
V_Dampf_nach_Komp_String:='ZU';
ELSE
V_Dampf_nach_Komp_String:='Offen';
END_IF;
IF V_Nach_WT  THEN
V_Nach_WT_String:='ZU';
ELSE
V_Nach_WT_String:='Offen';
END_IF;
IF V_Entlueftung_1 THEN
V_Entlueftung_1_String:='ZU';
ELSE
V_Entlueftung_1_String:='Offen';
END_IF;
IF V_Entlueftung_2  THEN
V_Entlueftung_2_String:='ZU';
ELSE
V_Entlueftung_2_String:='Offen';
END_IF;
IF V_Global_Res_3 THEN
V_Global_Res_3_String:='ZU';
ELSE
V_Global_Res_3_String:='Offen';
END_IF;
IF V_Global_Res_4 THEN
V_Global_Res_4_String:='Offen';
ELSE
V_Global_Res_4_String:='ZU';
END_IF;
IF V_Global_Res_5 THEN
V_Global_Res_5_String:='ZU';
ELSE
V_Global_Res_5_String:='Offen';
END_IF;






(* Dies müsste ev. in die Manu-Schlaufe, falls der Auto-Betrieb aktiviert wird!!*)


(*NO*)


IF V_Dampf_nach_Komp_Reset THEN V_Dampf_nach_Komp_Sequence:=FALSE; END_IF;
SR1(SET1:= V_Dampf_nach_Komp_manu OR V_Dampf_nach_Komp_Sequence  , RESET:=V_Dampf_nach_Komp_Reset  OR V_Dampf_nach_Komp_Reset_Sequence , Q1=> V_Dampf_nach_Komp_negiert );

(*Da dies ein 3/2-Wege ventil ist muss immer eine Seite des Ventils angesteuert sein, darum die negierte variable*)
V_Dampf_nach_Komp:= NOT V_Dampf_nach_Komp_negiert;

(*NO*)
IF V_Nach_WT_Reset  THEN V_Nach_WT_Sequence:=FALSE; END_IF;
SR2(SET1:= V_Nach_WT_manu OR V_Nach_WT_Sequence  , RESET:=V_Nach_WT_Reset  OR V_Nach_WT_Reset_Sequence , Q1=> V_Nach_WT_negiert);
V_Nach_WT :=NOT V_Nach_WT_negiert;


(*NO*)
IF V_Entlueftung_1_Reset THEN V_Entlueftung_1_Sequence:=FALSE; END_IF;
SR3(SET1:= V_Entlueftung_1_manu OR V_Entlueftung_1_Sequence  , RESET:=V_Entlueftung_1_Reset OR V_Entlueftung_1_Reset_Sequence , Q1=> V_Entlueftung_1_negiert );
V_Entlueftung_1:=NOT V_Entlueftung_1_negiert;


(*NO*)
IF V_Entlueftung_2_Reset THEN V_Entlueftung_2_Sequence:=FALSE; END_IF;
SR4(SET1:= V_Entlueftung_2_manu  OR V_Entlueftung_2_Sequence  , RESET:=V_Entlueftung_2_Reset OR V_Entlueftung_2_Reset_Sequence , Q1=> V_Entlueftung_2 );
V_Entlueftung_2_negiert:=NOT V_Entlueftung_2;

(*NO*)
IF V_Global_Res_3_Reset  THEN V_Global_Res_3_Sequence:=FALSE; END_IF;
SR5(SET1:= V_Global_Res_3_manu  OR V_Global_Res_3_Sequence  , RESET:=V_Global_Res_3_Reset  OR V_Global_Res_3_Reset_Sequence, Q1=> V_Global_Res_3 );
V_Global_Res_3_negiert:=NOT V_Global_Res_3;


(*NC*)
IF V_Global_Res_4_Reset  THEN V_Global_Res_4_Sequence:=FALSE; END_IF;
SR6(SET1:= V_Global_Res_4_manu  OR V_Global_Res_4_Sequence  , RESET:= V_Global_Res_4_Reset  OR  V_Global_Res_4_Reset_Sequence, Q1=>  V_Global_Res_4 );
V_Global_Res_4_negiert:=NOT  V_Global_Res_4;


(*NO*)
IF V_Global_Res_5_Reset THEN V_Global_Res_5_Sequence:=FALSE; END_IF;
SR7(SET1:= V_Global_Res_5_manu OR V_Global_Res_5_Sequence  , RESET:=V_Global_Res_5_Reset  OR V_Global_Res_5_Reset_Sequence , Q1=> V_Global_Res_5 );
V_Global_Res_5_negiert:=NOT V_Global_Res_5;











F_TRIG2(CLK:=V_Dampf_nach_Komp_Sequence );
IF F_TRIG2.Q THEN
V_Dampf_nach_Komp_Reset_Sequence :=TRUE;
ELSE
V_Dampf_nach_Komp_Reset_Sequence :=FALSE;
END_IF;

F_TRIG3(CLK:=V_Nach_WT_Sequence );
IF F_TRIG3.Q THEN
V_Nach_WT_Reset_Sequence :=TRUE;
ELSE
V_Nach_WT_Reset_Sequence :=FALSE;
END_IF;

F_TRIG4(CLK:=V_Entlueftung_1_Sequence );
IF F_TRIG4.Q THEN
V_Entlueftung_1_Reset_Sequence :=TRUE;
ELSE
V_Entlueftung_1_Reset_Sequence :=FALSE;
END_IF;

F_TRIG5(CLK:=V_Entlueftung_2_Sequence );
IF F_TRIG5.Q THEN
V_Entlueftung_2_Reset_Sequence :=TRUE;
ELSE
V_Entlueftung_2_Reset_Sequence :=FALSE;
END_IF;

F_TRIG6(CLK:=V_Global_Res_3_Sequence );
IF F_TRIG6.Q THEN
V_Global_Res_3_Reset_Sequence :=TRUE;
ELSE
V_Global_Res_3_Reset_Sequence :=FALSE;
END_IF;


F_TRIG7(CLK:=V_Global_Res_4_Sequence );
IF F_TRIG7.Q THEN
V_Global_Res_4_Reset_Sequence :=TRUE;
ELSE
V_Global_Res_4_Reset_Sequence :=FALSE;
END_IF;

F_TRIG8(CLK:=V_Global_Res_5_Sequence );
IF F_TRIG8.Q THEN
V_Global_Res_5_Reset_Sequence :=TRUE;
ELSE
V_Global_Res_5_Reset_Sequence :=FALSE;
END_IF;









V_Dampf_nach_Komp_Sequence:=VE_K2_71;
V_Nach_WT_Sequence:=VE_K2_73;
(*
V_Entlueftung_1_Sequence:=VE_K3_13;
V_Entlueftung_2_Sequence:=VE_K3_14;
V_Global_Res_3_Sequence:=VE_K3_18;
V_Global_Res_4_Sequence:=VE_K3_19;
V_Global_Res_5_Sequence:=VE_K3_20;
*)






(*Signalsäule Test*)

LED_RED_OUT:= LED_RED_VISU OR LED_RED_auto;
LED_green_OUT:= LED_green_VISU OR LED_green_auto;
LED_yellow_OUT:= LED_yellow_VISU OR LED_yellow_auto;
LED_white_OUT:= LED_white_VISU OR LED_white_auto;


IF counup_Array >= 10000 THEN
	counup_Array:=0;
	aArray_Histogram[0]:=0;
	aArray_Histogram[1]:=0;
	aArray_Histogram[2]:=0;
	aArray_Histogram[3]:=0;
	aArray_Histogram[4]:=0;
	aArray_Histogram[5]:=0;

	
END_IF;

counup_Array:=counup_Array+1;

counup_Array_OUT:=counup_Array/100;

counup_Array:=counup_Array+counup_Array;
aArray_Histogram[0]:=counup_Array_OUT+11;
aArray_Histogram[1]:=counup_Array_OUT+22;
aArray_Histogram[2]:=counup_Array_OUT+33;
aArray_Histogram[3]:=counup_Array_OUT+44;
aArray_Histogram[4]:=counup_Array_OUT+55;
aArray_Histogram[5]:=counup_Array_OUT+66;







(*Scope-View ZuweisunG


Da die anzahl der Var. welche beim Einlesen vom Scope view2 beschränkt ist, wurde eine zweite globale Var-Tabelle (GVL_1) deklariert
Diese dort einhaltenen Vars werden mit dem selben Prfix GVL_1.xy aufgerufen. Die Anzahl dort enthaltenen vars sind einiges weniger und deshalb können diese Infos vom Scope eingelesen werden*)

